	{attribute 'TcIecLibraryType'}
	{attribute 'external_name' := 'F_VN_CreateStaModel_GUID_E57A5C51_9E90_B9A1_5702_3D94CC195C09'}
	(* Create a Simplified TopoART neural network of the specified type. The initial reference count is set to one if a new model is created and kept, otherwise. Models of this type support on-line training (sample by sample), retraining, as well as scalar and vectorial predictions. It requires all input except class labels (i.e., samples and training outputs/predictions) to lie in the interval [0.0, 1.0]. The predictions of regressors need to be rescaled from the interval [0.0, 1.0] to their respective value range before usage. Depending on the parameter settings and the number of available training samples, repeated training with the same data may improve the results. Like other neural networks based on the Adaptive Resonance Theory (ART), Simplified TopoART neural networks are not prone to catastrophic inference and patricularly well-suited to incremental learning tasks. *)
	FUNCTION F_VN_CreateStaModel : HRESULT
	VAR_INPUT
		ipMlModel	:	REFERENCE TO ITcVnMlModel;	(* Returns the created model (Non-zero interface pointers are reused.) *)
		eStaType	:	ETcVnSta;	(* Simpified TopoART model type *)
		fRho	:	LREAL;	(* Vigilance parameter (controls the number of neurons that are inserted and the maximum size of the formed categories; valid range: [0.0, 1.0]; suggested range: [0.8, 1.0)) *)
		hrPrev	:	HRESULT;	(* HRESULT indicating the result of previous operations (If SUCCEEDED(hrPrev) equals false, no operation is executed.) *)
	END_VAR

END_FUNCTION

// Functions/Machine Learning/F_VN_CreateStaModelExp

	{attribute 'TcIecLibraryType'}
	{attribute 'external_name' := 'F_VN_CreateStaModelExp_GUID_8BD6F583_6D68_B761_42B8_60DD8485D486'}
	(* Create a Simplified TopoART neural network of the specified type. The initial reference count is set to one if a new model is created and kept, otherwise. Models of this type support on-line training (sample by sample), retraining, as well as scalar and vectorial predictions. It requires all input except class labels (i.e., samples and training outputs/predictions) to lie in the interval [0.0, 1.0]. The predictions of regressors need to be rescaled from the interval [0.0, 1.0] to their respective value range before usage. Depending on the parameter settings and the number of available training samples, repeated training with the same data may improve the results. Like other neural networks based on the Adaptive Resonance Theory (ART), Simplified TopoART neural networks are not prone to catastrophic inference and patricularly well-suited to incremental learning tasks. (expert function) *)
	FUNCTION F_VN_CreateStaModelExp : HRESULT
	VAR_INPUT
		ipMlModel	:	REFERENCE TO ITcVnMlModel;	(* Returns the created model (Non-zero interface pointers are reused.) *)
		eStaType	:	ETcVnSta;	(* Simpified TopoART model type *)
		fRho	:	LREAL;	(* Vigilance parameter (controls the number of neurons that are inserted and the maximum size of the formed categories; valid range: [0.0, 1.0]; suggested range: [0.8, 1.0)) *)
		nNu	:	UDINT;	(* Number of neurons used for classification and prediction (must be larger than or equal to 1; suggested range: [1, 10); default: 3) *)
		bDoublePrecision	:	BOOL;	(* If true, the model is generated with double precision (LREAL) instead of single precision (REAL). (default: FALSE) *)
		hrPrev	:	HRESULT;	(* HRESULT indicating the result of previous operations (If SUCCEEDED(hrPrev) equals false, no operation is executed.) *)
	END_VAR

END_FUNCTION

// Functions/Machine Learning/F_VN_CreateStaModelExp2

	{attribute 'TcIecLibraryType'}
	{attribute 'external_name' := 'F_VN_CreateStaModelExp2_GUID_374514C7_49DC_B14C_5A87_3ADAC4837261'}
	(* Create a Simplified TopoART neural network of the specified type. The initial reference count is set to one if a new model is created and kept, otherwise. Models of this type support on-line training (sample by sample), retraining, as well as scalar and vectorial predictions. It requires all input except class labels (i.e., samples and training outputs/predictions) to lie in the interval [0.0, 1.0]. The predictions of regressors need to be rescaled from the interval [0.0, 1.0] to their respective value range before usage. Depending on the parameter settings and the number of available training samples, repeated training with the same data may improve the results. Like other neural networks based on the Adaptive Resonance Theory (ART), Simplified TopoART neural networks are not prone to catastrophic inference and patricularly well-suited to incremental learning tasks. (additional expert function providing parameters for fine-tuning and noise reduction) *)
	FUNCTION F_VN_CreateStaModelExp2 : HRESULT
	VAR_INPUT
		ipMlModel	:	REFERENCE TO ITcVnMlModel;	(* Returns the created model (Non-zero interface pointers are reused.) *)
		eStaType	:	ETcVnSta;	(* Simpified TopoART model type *)
		fRho	:	LREAL;	(* Vigilance parameter (controls the number of neurons that are inserted and the maximum size of the formed categories; valid range: [0.0, 1.0]; suggested range: [0.8, 1.0)) *)
		nNu	:	UDINT;	(* Number of neurons used for classification and prediction (must be larger than or equal to 1; suggested range: [1, 10); default: 3) *)
		bDoublePrecision	:	BOOL;	(* If true, the model is generated with double precision (LREAL) instead of single precision (REAL). (default: FALSE) *)
		fBetaSbm	:	LREAL;	(* Learning rate of the second best-matching neuron (learning the second best-matching neuron keeps related categories closer together and might improve the results but may require a higher number of neurons and training runs; a value of 0.0 disables learning of the second best-matching neuron; valid range: [0.0, 1.0]; suggested range: [0.0, 0.5]); default: 0.0 *)
		nPhi	:	UDINT;	(* Number of samples a neuron must have learnt to become permanent (required for noise reduction; works in conjunction with nTau; must be larger than or equal to 1; higher values intensify noise reduction; a value of 1 disables removal of neuron candidates; default: 1) *)
		nTau	:	UDINT;	(* Number of learning steps after which node removal is performed (required for noise reduction; works in conjunction with nPhi; must be large enough to allow neuron candidates representing non-noise samples to become the best-matching neuron at least nPhi times before node removal; default: 100) *)
		hrPrev	:	HRESULT;	(* HRESULT indicating the result of previous operations (If SUCCEEDED(hrPrev) equals false, no operation is executed.) *)
	END_VAR

END_FUNCTION

// Functions/Machine Learning/F_VN_CreateSvmModel

	{attribute 'TcIecLibraryType'}
	{attribute 'external_name' := 'F_VN_CreateSvmModel_GUID_8D17BE1A_260C_B8D5_796F_11D521846FD9'}
	(* Create an SVM model of the specified type. The initial reference count is set to one if a new model is created and kept, otherwise. Models of this type neither support on-line training (sample by sample) nor retraining. Predictions can only be scalar. *)
	FUNCTION F_VN_CreateSvmModel : HRESULT
	VAR_INPUT
		ipMlModel	:	REFERENCE TO ITcVnMlModel;	(* Returns the created model (Non-zero interface pointers are reused.) *)
		eSvmType	:	ETcVnSvm;	(* SVM model type *)
		fC	:	LREAL;	(* Parameter C (required for TCVN_SVM_C_CLASSIFIER, TCVN_SVM_EPS_REGRESSOR, and TCVN_SVM_NU_REGRESSOR; ignored otherwise) *)
		fNu	:	LREAL;	(* Parameter nu (required for TCVN_SVM_NU_CLASSIFIER, TCVN_SVM_NOVELTY_DETECTOR, and TCVN_SVM_NU_REGRESSOR; ignored otherwise) *)
		fP	:	LREAL;	(* Parameter p (required for TCVN_SVM_EPS_REGRESSOR; ignored otherwise) *)
		eKernelType	:	ETcVnSvmKernelType;	(* Kernel type *)
		fGamma	:	LREAL;	(* Parameter gamma (used by polynomial, RBF, sigmoid, and chi-squared kernels; ignored otherwise) *)
		fCoef0	:	LREAL;	(* parameter coef0 (used by polynomial and sigmoid kernels; ignored otherwise) *)
		fDegree	:	LREAL;	(* Degree (used by polynomial kernels; ignored otherwise) *)
		hrPrev	:	HRESULT;	(* HRESULT indicating the result of previous operations (If SUCCEEDED(hrPrev) equals false, no operation is executed.) *)
	END_VAR

END_FUNCTION

// Functions/Machine Learning/F_VN_CreateSvmModelExp

	{attribute 'TcIecLibraryType'}
	{attribute 'external_name' := 'F_VN_CreateSvmModelExp_GUID_80022415_75F2_B05A_48A0_04DE64383B9C'}
	(* Create an SVM model of the specified type. The initial reference count is set to one if a new model is created and kept, otherwise. Models of this type neither support on-line training (sample by sample) nor retraining. Predictions can only be scalar. (expert function) *)
	FUNCTION F_VN_CreateSvmModelExp : HRESULT
	VAR_INPUT
		ipMlModel	:	REFERENCE TO ITcVnMlModel;	(* Returns the created model (Non-zero interface pointers are reused.) *)
		eSvmType	:	ETcVnSvm;	(* SVM model type *)
		fC	:	LREAL;	(* Parameter C (required for TCVN_SVM_C_CLASSIFIER, TCVN_SVM_EPS_REGRESSOR, and TCVN_SVM_NU_REGRESSOR; ignored otherwise) *)
		fNu	:	LREAL;	(* Parameter nu (required for TCVN_SVM_NU_CLASSIFIER, TCVN_SVM_NOVELTY_DETECTOR, and TCVN_SVM_NU_REGRESSOR; ignored otherwise) *)
		fP	:	LREAL;	(* Parameter p (required for TCVN_SVM_EPS_REGRESSOR; ignored otherwise) *)
		eKernelType	:	ETcVnSvmKernelType;	(* Kernel type *)
		fGamma	:	LREAL;	(* Parameter gamma (used by polynomial, RBF, sigmoid, and chi-squared kernels; ignored otherwise) *)
		fCoef0	:	LREAL;	(* Parameter coef0 (used by polynomial and sigmoid kernels; ignored otherwise) *)
		fDegree	:	LREAL;	(* Degree (used by polynomial kernels; ignored otherwise) *)
		nMaxIterations	:	UDINT;	(* Maximum number of iterations (disabled if it equals 0 and fEpsilon is different from 0.0; triggers the usage of the default value of 100000 if nMaxIterations and fEpsilon equal 0) *)
		fEpsilon	:	LREAL;	(* Maximum allowed difference of the error between two successive iterations (disabled if it equals 0.0 and nMaxIterations is different from 0; triggers the usage of the default value of 0.00001 if nMaxIterations and fEpsilon equal 0) *)
		hrPrev	:	HRESULT;	(* HRESULT indicating the result of previous operations (If SUCCEEDED(hrPrev) equals false, no operation is executed.) *)
	END_VAR

END_FUNCTION

// Functions/Machine Learning/F_VN_CreateSvmModelExp2

	{attribute 'TcIecLibraryType'}
	{attribute 'external_name' := 'F_VN_CreateSvmModelExp2_GUID_84CA59A5_8507_BAA1_5BD6_0739A483F2C9'}
	(* Create an SVM model of the specified type. The initial reference count is set to one if a new model is created and kept, otherwise. Models of this type neither support on-line training (sample by sample) nor retraining. Predictions can only be scalar. (additional expert function for C support vector classifiers) *)
	FUNCTION F_VN_CreateSvmModelExp2 : HRESULT
	VAR_INPUT
		ipMlModel	:	REFERENCE TO ITcVnMlModel;	(* Returns the created model (Non-zero interface pointers are reused.) *)
		eSvmType	:	ETcVnSvm;	(* SVM model type *)
		fC	:	LREAL;	(* Parameter C (required for TCVN_SVM_C_CLASSIFIER, TCVN_SVM_EPS_REGRESSOR, and TCVN_SVM_NU_REGRESSOR; ignored otherwise) *)
		fNu	:	LREAL;	(* Parameter nu (required for TCVN_SVM_NU_CLASSIFIER, TCVN_SVM_NOVELTY_DETECTOR, and TCVN_SVM_NU_REGRESSOR; ignored otherwise) *)
		fP	:	LREAL;	(* Parameter p (required for TCVN_SVM_EPS_REGRESSOR; ignored otherwise) *)
		eKernelType	:	ETcVnSvmKernelType;	(* Kernel type *)
		fGamma	:	LREAL;	(* Parameter gamma (used by polynomial, RBF, sigmoid, and chi-squared kernels; ignored otherwise) *)
		fCoef0	:	LREAL;	(* Parameter coef0 (used by polynomial and sigmoid kernels; ignored otherwise) *)
		fDegree	:	LREAL;	(* Degree (used by polynomial kernels; ignored otherwise) *)
		nMaxIterations	:	UDINT;	(* Maximum number of iterations (disabled if it equals 0 and fEpsilon is different from 0.0; triggers the usage of the default value of 100000 if nMaxIterations and fEpsilon equal 0) *)
		fEpsilon	:	LREAL;	(* Maximum allowed difference of the error between two successive iterations (disabled if it equals 0.0 and nMaxIterations is different from 0; triggers the usage of the default value of 0.00001 if nMaxIterations and fEpsilon equal 0) *)
		ipClassWeights	:	ITcVnContainer;	(* Class weights (ContainerType_Vector_REAL or ContainerType_Vector_LREAL; only valid if eSvmType equals TCVN_SVM_C_CLASSIFIER; optional, set to 0 if not required or not allowed; default: 0) *)
		hrPrev	:	HRESULT;	(* HRESULT indicating the result of previous operations (If SUCCEEDED(hrPrev) equals false, no operation is executed.) *)
	END_VAR

END_FUNCTION

// Functions/Machine Learning/F_VN_CreateSvmSgdClassifier

	{attribute 'TcIecLibraryType'}
	{attribute 'external_name' := 'F_VN_CreateSvmSgdClassifier_GUID_22F18F98_6803_BC91_601C_6D905DB53F12'}
	(* Create a linear SVM classifier using stochastic gradient descent for training. The initial reference count is set to one if a new model is created and kept, otherwise. This SVM classifier is only applicable to binary classification problems. It learns a separating hyperplane between a class with label -1 and a class with label 1. These class labels are predefined. For training, any positive class labels are mapped to 1 and any negative class labels are mapped to -1. Models of this type neither support on-line training (sample by sample) nor retraining. *)
	FUNCTION F_VN_CreateSvmSgdClassifier : HRESULT
	VAR_INPUT
		ipMlModel	:	REFERENCE TO ITcVnMlModel;	(* Returns the created model (Non-zero interface pointers are reused.) *)
		hrPrev	:	HRESULT;	(* HRESULT indicating the result of previous operations (If SUCCEEDED(hrPrev) equals false, no operation is executed.) *)
	END_VAR

END_FUNCTION

// Functions/Machine Learning/F_VN_CreateSvmSgdClassifierExp

	{attribute 'TcIecLibraryType'}
	{attribute 'external_name' := 'F_VN_CreateSvmSgdClassifierExp_GUID_DE6E86CE_13B3_BF4B_4F7F_D5DFEC535232'}
	(* Create a linear SVM classifier using stochastic gradient descent for training. The initial reference count is set to one if a new model is created and kept, otherwise. This SVM classifier is only applicable to binary classification problems. It learns a separating hyperplane between a class with label -1 and a class with label 1. These class labels are predefined. For training, any positive class labels are mapped to 1 and any negative class labels are mapped to -1. Models of this type neither support on-line training (sample by sample) nor retraining. (expert function) *)
	FUNCTION F_VN_CreateSvmSgdClassifierExp : HRESULT
	VAR_INPUT
		ipMlModel	:	REFERENCE TO ITcVnMlModel;	(* Returns the created model (Non-zero interface pointers are reused.) *)
		eType	:	ETcVnSvmSgdClassifierType;	(* Learning algorithm type (default: TCVN_SSCT_ASGD) *)
		eMarginType	:	ETcVnSvmSgdClassifierMarginType;	(* Margin type (default: TCVN_SSCMT_SOFT_MARGIN) *)
		fMarginRegularization	:	REAL;	(* Margin regularization parameter (default: 0.00001) *)
		fInitialStepSize	:	REAL;	(* Initial step size (default: 0.05) *)
		fStepDecreasingPower	:	REAL;	(* Power parameter (default: 0.75) *)
		nMaxIterations	:	UDINT;	(* Maximum number of iterations (disabled if it equals 0 and fEpsilon is different from 0.0; triggers the usage of the default value of 100000 if nMaxIterations and fEpsilon equal 0) *)
		fEpsilon	:	LREAL;	(* Maximum allowed difference of the error between two successive iterations (disabled if it equals 0.0 and nMaxIterations is different from 0; triggers the usage of the default value of 0.00001 if nMaxIterations and fEpsilon equal 0) *)
		hrPrev	:	HRESULT;	(* HRESULT indicating the result of previous operations (If SUCCEEDED(hrPrev) equals false, no operation is executed.) *)
	END_VAR

END_FUNCTION

// Functions/Machine Learning/F_VN_FeatureTransform

	{attribute 'TcIecLibraryType'}
	{attribute 'external_name' := 'F_VN_FeatureTransform_GUID_2D180149_1314_B2CD_6D03_B45D7BAFFB33'}
	(* Apply a feature transform to one or more sample(s). *)
	FUNCTION F_VN_FeatureTransform : HRESULT
	VAR_INPUT
		ipFeatureTransform	:	ITcVnMlModel;	(* Feature transform instance to be used *)
		ipSamples	:	ITcUnknown;	(* Container holding one or more of input sample(s) (ContainerType_Vector_REAL, ContainerType_Vector_LREAL, ContainerType_Vector_Vector_REAL, or ContainerType_Vector_Vector_LREAL) *)
		pipTransformed	:	POINTER TO ITcUnknown;	(* Returns the transformed sample(s) using the same type like ipSamples *)
		hrPrev	:	HRESULT;	(* HRESULT indicating the result of previous operations (If SUCCEEDED(hrPrev) equals false, no operation is executed.) *)
	END_VAR

END_FUNCTION

// Functions/Machine Learning/F_VN_GetBatchClusters

	{attribute 'TcIecLibraryType'}
	{attribute 'external_name' := 'F_VN_GetBatchClusters_GUID_B991822A_20BF_BAE1_5901_CECBAF3E4795'}
	(* Get the IDs of the best-matching clusters of a batch of samples. *)
	FUNCTION F_VN_GetBatchClusters : HRESULT
	VAR_INPUT
		ipClusterer	:	ITcVnMlModel;	(* Clusterer to be used *)
		ipSamples	:	ITcUnknown;	(* Container holding a batch of input samples (ContainerType_Vector_Vector_REAL or ContainerType_Vector_Vector_LREAL) *)
		ipClusters	:	REFERENCE TO ITcVnContainer;	(* Returns the cluster IDs (ContainerType_Vector_DINT) *)
		hrPrev	:	HRESULT;	(* HRESULT indicating the result of previous operations (If SUCCEEDED(hrPrev) equals false, no operation is executed.) *)
	END_VAR

END_FUNCTION

// Functions/Machine Learning/F_VN_GetBatchClustersExp

	{attribute 'TcIecLibraryType'}
	{attribute 'external_name' := 'F_VN_GetBatchClustersExp_GUID_01381543_FF2C_BDB4_623D_753D989F9781'}
	(* Get the IDs of the best-matching clusters of a batch of samples. *)
	FUNCTION F_VN_GetBatchClustersExp : HRESULT
	VAR_INPUT
		ipClusterer	:	ITcVnMlModel;	(* Clusterer to be used *)
		ipSamples	:	ITcUnknown;	(* Container holding a batch of input samples (ContainerType_Vector_Vector_REAL or ContainerType_Vector_Vector_LREAL) *)
		ipClusters	:	REFERENCE TO ITcVnContainer;	(* Returns the cluster IDs (ContainerType_Vector_DINT) *)
		ipNovelties	:	REFERENCE TO ITcVnContainer;	(* Returns the degree of novelty (0.0 if a sample is completely known; > 0.0 otherwise) of each sample (ContainerType_Vector_REAL; optional, set to 0 if not required) *)
		hrPrev	:	HRESULT;	(* HRESULT indicating the result of previous operations (If SUCCEEDED(hrPrev) equals false, no operation is executed.) *)
	END_VAR

END_FUNCTION

// Functions/Machine Learning/F_VN_GetBatchNovelties

	{attribute 'TcIecLibraryType'}
	{attribute 'external_name' := 'F_VN_GetBatchNovelties_GUID_97240524_1B64_B7E2_556C_1ACF30F41F39'}
	(* Get the degree of novelty of multiple samples. *)
	FUNCTION F_VN_GetBatchNovelties : HRESULT
	VAR_INPUT
		ipNoveltyDetector	:	ITcVnMlModel;	(* Novelty detector to be used *)
		ipSamples	:	ITcUnknown;	(* Container holding a batch of input samples (ContainerType_Vector_Vector_REAL or ContainerType_Vector_Vector_LREAL) *)
		ipNovelties	:	REFERENCE TO ITcVnContainer;	(* Returns the degree of novelty (0.0 if a sample is completely known; > 0.0 otherwise) of each sample (ContainerType_Vector_REAL) *)
		hrPrev	:	HRESULT;	(* HRESULT indicating the result of previous operations (If SUCCEEDED(hrPrev) equals false, no operation is executed.) *)
	END_VAR

END_FUNCTION

// Functions/Machine Learning/F_VN_GetClusterCenter

	{attribute 'TcIecLibraryType'}
	{attribute 'external_name' := 'F_VN_GetClusterCenter_GUID_E4931504_8DC6_B6D3_5D5D_2EFA9234F477'}
	(* Get the center of a cluster. *)
	FUNCTION F_VN_GetClusterCenter : HRESULT
	VAR_INPUT
		ipClusterer	:	ITcVnMlModel;	(* Clusterer to be used *)
		nCluster	:	DINT;	(* Cluster ID of the cluster the center of which is requested *)
		ipCenter	:	REFERENCE TO ITcVnContainer;	(* Returns the cluster center (ContainerType_Vector_REAL or ContainerType_Vector_LREAL depending on the floating point type internally used by the clusterer) *)
		hrPrev	:	HRESULT;	(* HRESULT indicating the result of previous operations (If SUCCEEDED(hrPrev) equals false, no operation is executed.) *)
	END_VAR

END_FUNCTION

// Functions/Machine Learning/F_VN_GetClusterNum

	{attribute 'TcIecLibraryType'}
	{attribute 'external_name' := 'F_VN_GetClusterNum_GUID_BF90D70E_F34B_BD2C_7F4D_80A10CF6A5F4'}
	(* Get the number of clusters used by this clusterer. *)
	FUNCTION F_VN_GetClusterNum : HRESULT
	VAR_INPUT
		ipClusterer	:	ITcVnMlModel;	(* Clusterer to be used *)
	END_VAR
	VAR_IN_OUT
		nClusterNum	:	ULINT;	(* Returns the number of clusters *)
	END_VAR
	VAR_INPUT
		hrPrev	:	HRESULT;	(* HRESULT indicating the result of previous operations (If SUCCEEDED(hrPrev) equals false, no operation is executed.) *)
	END_VAR

END_FUNCTION

// Functions/Machine Learning/F_VN_GetFeatureScales

	{attribute 'TcIecLibraryType'}
	{attribute 'external_name' := 'F_VN_GetFeatureScales_GUID_152933F4_9817_B6E4_5FDD_5FA5A50599FB'}
	(* Calculate the scaling parameters for each feature in the input samples based on the scaling type. *)
	FUNCTION F_VN_GetFeatureScales : HRESULT
	VAR_INPUT
		ipSamples	:	ITcVnContainer;	(* Container holding input sample(s) (ContainerType_Vector_REAL, ContainerType_Vector_LREAL, ContainerType_Vector_Vector_REAL or ContainerType_Vector_Vector_LREAL) *)
		ipScales	:	REFERENCE TO ITcVnContainer;	(* Returns a container with the scaling parameters for each feature (Vector_REAL or Vector_LREAL depending on the type of ipSamples). *)
		eFeatureScalingType	:	ETcVnFeatureScalingType;	(* Feature scaling type *)
		hrPrev	:	HRESULT;	(* HRESULT indicating the result of previous operations (If SUCCEEDED(hrPrev) equals false, no operation is executed.) *)
	END_VAR

END_FUNCTION

// Functions/Machine Learning/F_VN_GetSampleCluster

	{attribute 'TcIecLibraryType'}
	{attribute 'external_name' := 'F_VN_GetSampleCluster_GUID_D9EDADE6_09DF_BF79_401D_9EFAF11AC262'}
	(* Get the ID of the best-matching cluster of a single sample. *)
	FUNCTION F_VN_GetSampleCluster : HRESULT
	VAR_INPUT
		ipClusterer	:	ITcVnMlModel;	(* Clusterer to be used *)
		ipSample	:	ITcUnknown;	(* Container holding a single input sample (ContainerType_Vector_REAL or ContainerType_Vector_LREAL) *)
	END_VAR
	VAR_IN_OUT
		nCluster	:	DINT;	(* Returns the ID of the cluster the sample has been assigned to *)
	END_VAR
	VAR_INPUT
		hrPrev	:	HRESULT;	(* HRESULT indicating the result of previous operations (If SUCCEEDED(hrPrev) equals false, no operation is executed.) *)
	END_VAR

END_FUNCTION

// Functions/Machine Learning/F_VN_GetSampleClusterExp

	{attribute 'TcIecLibraryType'}
	{attribute 'external_name' := 'F_VN_GetSampleClusterExp_GUID_DF68DB58_441A_B462_5F9C_8B8B5A8B453F'}
	(* Get the ID of the best-matching cluster of a single sample. (expert function) *)
	FUNCTION F_VN_GetSampleClusterExp : HRESULT
	VAR_INPUT
		ipClusterer	:	ITcVnMlModel;	(* Clusterer to be used *)
		ipSample	:	ITcUnknown;	(* Container holding a single input sample (ContainerType_Vector_REAL or ContainerType_Vector_LREAL) *)
	END_VAR
	VAR_IN_OUT
		nCluster	:	DINT;	(* Returns the ID of the cluster the sample has been assigned to *)
	END_VAR
	VAR_INPUT
		fNovelty	:	REFERENCE TO REAL;	(* Returns the degree of novelty (0.0 if a sample is completely known; > 0.0 otherwise) of the presented sample (optional, set to 0 if not required) *)
		hrPrev	:	HRESULT;	(* HRESULT indicating the result of previous operations (If SUCCEEDED(hrPrev) equals false, no operation is executed.) *)
	END_VAR

END_FUNCTION

// Functions/Machine Learning/F_VN_GetSampleNovelty

	{attribute 'TcIecLibraryType'}
	{attribute 'external_name' := 'F_VN_GetSampleNovelty_GUID_39A873D6_D903_BC16_5D0D_1737EA55271D'}
	(* Get the degree of novelty of a single sample. *)
	FUNCTION F_VN_GetSampleNovelty : HRESULT
	VAR_INPUT
		ipNoveltyDetector	:	ITcVnMlModel;	(* Novelty detector to be used *)
		ipSample	:	ITcUnknown;	(* Container holding a single input sample (ContainerType_Vector_REAL or ContainerType_Vector_LREAL) *)
	END_VAR
	VAR_IN_OUT
		fNovelty	:	REAL;	(* Returns the degree of novelty (0.0 if a sample is completely known; > 0.0 otherwise) of the presented sample *)
	END_VAR
	VAR_INPUT
		hrPrev	:	HRESULT;	(* HRESULT indicating the result of previous operations (If SUCCEEDED(hrPrev) equals false, no operation is executed.) *)
	END_VAR

END_FUNCTION

// Functions/Machine Learning/F_VN_InverseFeatureScaling

	{attribute 'TcIecLibraryType'}
	{attribute 'external_name' := 'F_VN_InverseFeatureScaling_GUID_FE8FDE22_64A6_B82E_5950_09F49A4CC796'}
	(* Apply the inverse of feature scaling to one or more sample(s). *)
	FUNCTION F_VN_InverseFeatureScaling : HRESULT
	VAR_INPUT
		ipSamples	:	ITcVnContainer;	(* Container holding one or more input sample(s) (ContainerType_Vector_REAL, ContainerType_Vector_LREAL, ContainerType_Vector_Vector_REAL, or ContainerType_Vector_Vector_LREAL) *)
		ipScales	:	ITcVnContainer;	(* Container with the scaling parameters of each feature (type ContainerType_Vector_REAL or ContainerType_Vector_LREAL). *)
		ipInverseSamples	:	REFERENCE TO ITcVnContainer;	(* Returns the inversed sample(s) using the scaling type and parameters of ipScales. It has the same type of ipSamples. If the same container ipSamples is used, the source data will be replaced. *)
		hrPrev	:	HRESULT;	(* HRESULT indicating the result of previous operations (If SUCCEEDED(hrPrev) equals false, no operation is executed.) *)
	END_VAR

END_FUNCTION

// Functions/Machine Learning/F_VN_InverseFeatureScaling_REAL

	{attribute 'TcIecLibraryType'}
	{attribute 'external_name' := 'F_VN_InverseFeatureScaling_REAL_GUID_1201C1F8_7D25_B625_41FC_0E90A3247281'}
	(* Apply the inverse of feature scaling to a single value. *)
	FUNCTION F_VN_InverseFeatureScaling_REAL : HRESULT
	VAR_INPUT
		fSample	:	REAL;	(* Sample value *)
		ipScales	:	ITcVnContainer;	(* Container with the scaling parameters of each feature (type ContainerType_Vector_REAL or ContainerType_Vector_LREAL). *)
	END_VAR
	VAR_IN_OUT
		fInverseSample	:	REAL;	(* Returns the inversed sample. *)
	END_VAR
	VAR_INPUT
		hrPrev	:	HRESULT;	(* HRESULT indicating the result of previous operations (If SUCCEEDED(hrPrev) equals false, no operation is executed.) *)
	END_VAR

END_FUNCTION

// Functions/Machine Learning/F_VN_InverseFeatureScalingExp

	{attribute 'TcIecLibraryType'}
	{attribute 'external_name' := 'F_VN_InverseFeatureScalingExp_GUID_6011A69B_BC3C_B4AD_6BA0_0FF48B427FDA'}
	(* Apply the inverse of feature scaling to one or more sample(s). [fA, fB] should be used if the scaling has been performed using TCVN_FST1_MINMAX with a predetermined output range.. (expert function) *)
	FUNCTION F_VN_InverseFeatureScalingExp : HRESULT
	VAR_INPUT
		ipSamples	:	ITcVnContainer;	(* Container holding one or more input sample(s) (ContainerType_Vector_REAL, ContainerType_Vector_LREAL, ContainerType_Vector_Vector_REAL, or ContainerType_Vector_Vector_LREAL) *)
		ipScales	:	ITcVnContainer;	(* Container with the scaling parameters of each feature (type ContainerType_Vector_REAL or ContainerType_Vector_LREAL). *)
		ipInverseSamples	:	REFERENCE TO ITcVnContainer;	(* Returns the inversed sample(s) using the scaling type and parameters of ipScales. It has the same type of ipSamples. If the same container ipSamples is used, the source data will be replaced. *)
		fA	:	LREAL;	(* represents the lower bound of the range for TCVN_FST1_MINMAX *)
		fB	:	LREAL;	(* represents the upper bound of the range for TCVN_FST1_MINMAX *)
		hrPrev	:	HRESULT;	(* HRESULT indicating the result of previous operations (If SUCCEEDED(hrPrev) equals false, no operation is executed.) *)
	END_VAR

END_FUNCTION

// Functions/Machine Learning/F_VN_InverseFeatureScalingExp_REAL

	{attribute 'TcIecLibraryType'}
	{attribute 'external_name' := 'F_VN_InverseFeatureScalingExp_REAL_GUID_C9B73D36_4564_B6F0_65B6_270F53192161'}
	(* Apply the inverse of feature scaling to a single value. [fA, fB] should be used if the scaling has been performed using TCVN_FST1_MINMAX with a predetermined output range. *)
	FUNCTION F_VN_InverseFeatureScalingExp_REAL : HRESULT
	VAR_INPUT
		fSample	:	REAL;	(* Sample value *)
		ipScales	:	ITcVnContainer;	(* Container with the scaling parameters of each feature (type ContainerType_Vector_REAL or ContainerType_Vector_LREAL). *)
	END_VAR
	VAR_IN_OUT
		fInverseSample	:	REAL;	(* Returns the inversed sample. *)
	END_VAR
	VAR_INPUT
		fA	:	LREAL;	(* represents the lower bound of the range for TCVN_FST1_MINMAX *)
		fB	:	LREAL;	(* represents the upper bound of the range for TCVN_FST1_MINMAX *)
		hrPrev	:	HRESULT;	(* HRESULT indicating the result of previous operations (If SUCCEEDED(hrPrev) equals false, no operation is executed.) *)
	END_VAR

END_FUNCTION

// Functions/Machine Learning/F_VN_InverseFeatureTransform

	{attribute 'TcIecLibraryType'}
	{attribute 'external_name' := 'F_VN_InverseFeatureTransform_GUID_36FA6EBF_2E20_B057_4C4D_1F432CD52CC5'}
	(* Apply an inverse feature transform to one or more sample(s). *)
	FUNCTION F_VN_InverseFeatureTransform : HRESULT
	VAR_INPUT
		ipFeatureTransform	:	ITcVnMlModel;	(* Feature transform instance to be used *)
		ipSamples	:	ITcUnknown;	(* Container holding one or more of input sample(s) (ContainerType_Vector_REAL, ContainerType_Vector_LREAL, ContainerType_Vector_Vector_REAL, or ContainerType_Vector_Vector_LREAL) *)
		pipTransformed	:	POINTER TO ITcUnknown;	(* Returns the transformed sample(s) using the same type like ipSamples *)
		hrPrev	:	HRESULT;	(* HRESULT indicating the result of previous operations (If SUCCEEDED(hrPrev) equals false, no operation is executed.) *)
	END_VAR

END_FUNCTION

// Functions/Machine Learning/F_VN_PredictBatch

	{attribute 'TcIecLibraryType'}
	{attribute 'external_name' := 'F_VN_PredictBatch_GUID_7D6AF5D3_F545_BA81_6792_DBF8D05FF13D'}
	(* Compute predictions for a batch of samples. *)
	FUNCTION F_VN_PredictBatch : HRESULT
	VAR_INPUT
		ipMlModel	:	ITcVnMlModel;	(* Classifier or regressor to be used *)
		ipSamples	:	ITcUnknown;	(* Container holding a batch of input samples (ContainerType_Vector_Vector_REAL or ContainerType_Vector_Vector_LREAL) *)
		ipPredictions	:	REFERENCE TO ITcVnContainer;	(* Returns the predicted outputs (depending on ipSamples; class labels (for classification, ContainerType_Vector_DINT) or real-valued predictions (for regression with scalar output, ContainerType_Vector_REAL or ContainerType_Vector_LREAL; for regression with vectorial output, ContainerType_Vector_Vector_REAL or ContainerType_Vector_Vector_LREAL)) *)
		hrPrev	:	HRESULT;	(* HRESULT indicating the result of previous operations (If SUCCEEDED(hrPrev) equals false, no operation is executed.) *)
	END_VAR

END_FUNCTION

// Functions/Machine Learning/F_VN_PredictBatchExp

	{attribute 'TcIecLibraryType'}
	{attribute 'external_name' := 'F_VN_PredictBatchExp_GUID_C38FEE18_09F7_BE98_52DE_06033125E4BC'}
	(* Compute predictions for a batch of samples. (expert function) *)
	FUNCTION F_VN_PredictBatchExp : HRESULT
	VAR_INPUT
		ipMlModel	:	ITcVnMlModel;	(* Classifier or regressor to be used *)
		ipSamples	:	ITcUnknown;	(* Container holding a batch of input samples (ContainerType_Vector_Vector_REAL or ContainerType_Vector_Vector_LREAL) *)
		ipPredictions	:	REFERENCE TO ITcVnContainer;	(* Returns the predicted outputs (depending on ipSamples; class labels (for classification, ContainerType_Vector_DINT) or real-valued predictions (for regression with scalar output, ContainerType_Vector_REAL or ContainerType_Vector_LREAL; for regression with vectorial output, ContainerType_Vector_Vector_REAL or ContainerType_Vector_Vector_LREAL)) *)
		ipNovelties	:	REFERENCE TO ITcVnContainer;	(* Returns the degree of novelty (0.0 if a sample is completely known; > 0.0 otherwise) of each sample (ContainerType_Vector_REAL; optional, set to 0 if not required) *)
		hrPrev	:	HRESULT;	(* HRESULT indicating the result of previous operations (If SUCCEEDED(hrPrev) equals false, no operation is executed.) *)
	END_VAR

END_FUNCTION

// Functions/Machine Learning/F_VN_PredictSampleClass

	{attribute 'TcIecLibraryType'}
	{attribute 'external_name' := 'F_VN_PredictSampleClass_GUID_4E1D7695_AD53_B95E_78AD_1EE49BFC5C71'}
	(* Classify a single sample. *)
	FUNCTION F_VN_PredictSampleClass : HRESULT
	VAR_INPUT
		ipClassifier	:	ITcVnMlModel;	(* Classifier to be used *)
		ipSample	:	ITcUnknown;	(* Container holding a single input sample (ContainerType_Vector_REAL or ContainerType_Vector_LREAL) *)
	END_VAR
	VAR_IN_OUT
		nClass	:	DINT;	(* Returns the classification result *)
	END_VAR
	VAR_INPUT
		hrPrev	:	HRESULT;	(* HRESULT indicating the result of previous operations (If SUCCEEDED(hrPrev) equals false, no operation is executed.) *)
	END_VAR

END_FUNCTION

// Functions/Machine Learning/F_VN_PredictSampleClassExp

	{attribute 'TcIecLibraryType'}
	{attribute 'external_name' := 'F_VN_PredictSampleClassExp_GUID_7AF8CE47_2D0D_B2AE_4405_566F1365D87E'}
	(* Classify a single sample. (expert function) *)
	FUNCTION F_VN_PredictSampleClassExp : HRESULT
	VAR_INPUT
		ipClassifier	:	ITcVnMlModel;	(* Classifier to be used *)
		ipSample	:	ITcUnknown;	(* Container holding a single input sample (ContainerType_Vector_REAL or ContainerType_Vector_LREAL) *)
	END_VAR
	VAR_IN_OUT
		nClass	:	DINT;	(* Returns the classification result *)
	END_VAR
	VAR_INPUT
		fNovelty	:	REFERENCE TO REAL;	(* Returns the degree of novelty (0.0 if a sample is completely known; > 0.0 otherwise) of the presented sample (optional, set to 0 if not required) *)
		hrPrev	:	HRESULT;	(* HRESULT indicating the result of previous operations (If SUCCEEDED(hrPrev) equals false, no operation is executed.) *)
	END_VAR

END_FUNCTION

// Functions/Machine Learning/F_VN_PredictSampleScalar

	{attribute 'TcIecLibraryType'}
	{attribute 'external_name' := 'F_VN_PredictSampleScalar_GUID_A0660891_3ED0_BD79_45C7_B847E30A9869'}
	(* Compute a scalar prediction for a single sample. *)
	FUNCTION F_VN_PredictSampleScalar : HRESULT
	VAR_INPUT
		ipRegressor	:	ITcVnMlModel;	(* Regressor to be used *)
		ipSample	:	ITcUnknown;	(* Container holding a single input sample (ContainerType_Vector_REAL or ContainerType_Vector_LREAL) *)
	END_VAR
	VAR_IN_OUT
		fPrediction	:	REAL;	(* Returns the predicted output *)
	END_VAR
	VAR_INPUT
		hrPrev	:	HRESULT;	(* HRESULT indicating the result of previous operations (If SUCCEEDED(hrPrev) equals false, no operation is executed.) *)
	END_VAR

END_FUNCTION

// Functions/Machine Learning/F_VN_PredictSampleScalarExp

	{attribute 'TcIecLibraryType'}
	{attribute 'external_name' := 'F_VN_PredictSampleScalarExp_GUID_32126386_2E2D_B430_66C6_B8A4437C5BD6'}
	(* Compute a scalar prediction for a single sample. (expert function) *)
	FUNCTION F_VN_PredictSampleScalarExp : HRESULT
	VAR_INPUT
		ipRegressor	:	ITcVnMlModel;	(* Regressor to be used *)
		ipSample	:	ITcUnknown;	(* Container holding a single input sample (ContainerType_Vector_REAL or ContainerType_Vector_LREAL) *)
	END_VAR
	VAR_IN_OUT
		fPrediction	:	REAL;	(* Returns the predicted output *)
	END_VAR
	VAR_INPUT
		fNovelty	:	REFERENCE TO REAL;	(* Returns the degree of novelty (0.0 if a sample is completely known; > 0.0 otherwise) of the presented sample (optional, set to 0 if not required) *)
		hrPrev	:	HRESULT;	(* HRESULT indicating the result of previous operations (If SUCCEEDED(hrPrev) equals false, no operation is executed.) *)
	END_VAR

END_FUNCTION

// Functions/Machine Learning/F_VN_PredictSampleVector

	{attribute 'TcIecLibraryType'}
	{attribute 'external_name' := 'F_VN_PredictSampleVector_GUID_1341F380_9576_B968_589D_54E9FDC95A1C'}
	(* Compute a vectorial prediction for a single sample. *)
	FUNCTION F_VN_PredictSampleVector : HRESULT
	VAR_INPUT
		ipRegressor	:	ITcVnMlModel;	(* Regressor to be used *)
		ipSample	:	ITcUnknown;	(* Container holding a single input sample (ContainerType_Vector_REAL or ContainerType_Vector_LREAL) *)
		ipPrediction	:	REFERENCE TO ITcVnContainer;	(* Returns the predicted output (ContainerType_Vector_REAL or ContainerType_Vector_LREAL, depending on ipSample) *)
		hrPrev	:	HRESULT;	(* HRESULT indicating the result of previous operations (If SUCCEEDED(hrPrev) equals false, no operation is executed.) *)
	END_VAR

END_FUNCTION

// Functions/Machine Learning/F_VN_PredictSampleVectorExp

	{attribute 'TcIecLibraryType'}
	{attribute 'external_name' := 'F_VN_PredictSampleVectorExp_GUID_031F0675_23FD_B293_640F_296778A8E4F6'}
	(* Compute a vectorial prediction for a single sample. (expert function) *)
	FUNCTION F_VN_PredictSampleVectorExp : HRESULT
	VAR_INPUT
		ipRegressor	:	ITcVnMlModel;	(* Regressor to be used *)
		ipSample	:	ITcUnknown;	(* Container holding a single input sample (ContainerType_Vector_REAL or ContainerType_Vector_LREAL) *)
		ipPrediction	:	REFERENCE TO ITcVnContainer;	(* Returns the predicted output (ContainerType_Vector_REAL or ContainerType_Vector_LREAL, depending on ipSample) *)
		fNovelty	:	REFERENCE TO REAL;	(* Returns the degree of novelty (0.0 if a sample is completely known; > 0.0 otherwise) of the presented sample (optional, set to 0 if not required) *)
		hrPrev	:	HRESULT;	(* HRESULT indicating the result of previous operations (If SUCCEEDED(hrPrev) equals false, no operation is executed.) *)
	END_VAR

END_FUNCTION

// Functions/Machine Learning/F_VN_FeatureScaling

	{attribute 'TcIecLibraryType'}
	{attribute 'external_name' := 'F_VN_FeatureScaling_GUID_9BD98239_4277_BFE9_7F08_2E1B5FF5F5E8'}
	(* Apply a feature scaling to one or more sample(s). *)
	FUNCTION F_VN_FeatureScaling : HRESULT
	VAR_INPUT
		ipSamples	:	ITcVnContainer;	(* Container holding one or more input sample(s) (ContainerType_Vector_REAL, ContainerType_Vector_LREAL, ContainerType_Vector_Vector_REAL, or ContainerType_Vector_Vector_LREAL) *)
		ipScales	:	ITcVnContainer;	(* Container with the scaling parameters of each feature (type ContainerType_Vector_REAL or ContainerType_Vector_LREAL). *)
		ipScaledSamples	:	REFERENCE TO ITcVnContainer;	(* Returns the scaled sample(s) using the same type like ipSamples. If the same container ipSamples is uesd, the source data will be replaced. *)
		hrPrev	:	HRESULT;	(* HRESULT indicating the result of previous operations (If SUCCEEDED(hrPrev) equals false, no operation is executed.) *)
	END_VAR

END_FUNCTION

// Functions/Machine Learning/F_VN_FeatureScalingExp

	{attribute 'TcIecLibraryType'}
	{attribute 'external_name' := 'F_VN_FeatureScalingExp_GUID_62DE1C89_F96E_B166_52C9_6230A4FA8FF4'}
	(* Apply a feature scaling to one or more sample(s) and get output range between [fA, fB] in the case of TCVN_FST1_MINMAX.  (expert function) *)
	FUNCTION F_VN_FeatureScalingExp : HRESULT
	VAR_INPUT
		ipSamples	:	ITcVnContainer;	(* Container holding one or more input sample(s) (ContainerType_Vector_REAL, ContainerType_Vector_LREAL, ContainerType_Vector_Vector_REAL, or ContainerType_Vector_Vector_LREAL) *)
		ipScales	:	ITcVnContainer;	(* Container with the scaling parameters of each feature (type ContainerType_Vector_REAL or ContainerType_Vector_LREAL). *)
		ipScaledSamples	:	REFERENCE TO ITcVnContainer;	(* Returns the scaled sample(s) using the same type like ipSamples. If the same container ipSamples is uesd, the source data will be replaced. *)
		fA	:	LREAL;	(* represents the lower bound of the range for TCVN_FST1_MINMAX *)
		fB	:	LREAL;	(* represents the upper bound of the range for TCVN_FST1_MINMAX *)
		hrPrev	:	HRESULT;	(* HRESULT indicating the result of previous operations (If SUCCEEDED(hrPrev) equals false, no operation is executed.) *)
	END_VAR

END_FUNCTION

// Functions/Machine Learning/F_VN_TrainBatch

	{attribute 'TcIecLibraryType'}
	{attribute 'external_name' := 'F_VN_TrainBatch_GUID_77947D56_1092_B041_6AD6_45459A0EDE0C'}
	(* Train a classifier, a clusterer, a novelty detector, or a regressor with a batch of samples. On-line trainable models are trained once with each sample. Depending on the application and the number of available training samples, repeated training of such models with the same data may improve the results. *)
	FUNCTION F_VN_TrainBatch : HRESULT
	VAR_INPUT
		ipMlModel	:	ITcVnMlModel;	(* Classifier, clusterer, novelty detector, or regressor to be used *)
		ipSamples	:	ITcUnknown;	(* Container holding a batch of input samples (ContainerType_Vector_Vector_REAL or ContainerType_Vector_Vector_LREAL) *)
		ipOutputs	:	ITcVnContainer;	(* Class labels (for classification, ContainerType_Vector_DINT) or target outputs (for regression with scalar output, ContainerType_Vector_REAL or ContainerType_Vector_LREAL; for regression with vectorial output, ContainerType_Vector_Vector_REAL or ContainerType_Vector_Vector_LREAL) to be learnt (must be 0 for clusterers and for novelty detectors) *)
		hrPrev	:	HRESULT;	(* HRESULT indicating the result of previous operations (If SUCCEEDED(hrPrev) equals false, no operation is executed.) *)
	END_VAR

END_FUNCTION

// Functions/Machine Learning/F_VN_TrainBatchClusters

	{attribute 'TcIecLibraryType'}
	{attribute 'external_name' := 'F_VN_TrainBatchClusters_GUID_23468B3D_3C92_B481_59BE_FD8A5A9CA9B1'}
	(* Train a clusterer with a batch of samples and return the IDs of the clusters the samples have been assigned to, if requested. On-line trainable clusterers are trained once with each sample. Depending on the application and the number of available training samples, repeated training of such models with the same data may improve the results. *)
	FUNCTION F_VN_TrainBatchClusters : HRESULT
	VAR_INPUT
		ipClusterer	:	ITcVnMlModel;	(* Clusterer to be used *)
		ipSamples	:	ITcUnknown;	(* Container holding a batch of input samples (ContainerType_Vector_Vector_REAL or ContainerType_Vector_Vector_LREAL) *)
		ipClusters	:	REFERENCE TO ITcVnContainer;	(* Returns the IDs of the clusters the samples have been assigned to (ContainerType_Vector_DINT; optional, set to 0 if not required) *)
		hrPrev	:	HRESULT;	(* HRESULT indicating the result of previous operations (If SUCCEEDED(hrPrev) equals false, no operation is executed.) *)
	END_VAR

END_FUNCTION

// Functions/Machine Learning/F_VN_TrainSample

	{attribute 'TcIecLibraryType'}
	{attribute 'external_name' := 'F_VN_TrainSample_GUID_6B0A2796_5FCD_B08B_5BD0_FF7775FE4207'}
	(* Train a clusterer or a novelty detector with a single sample. *)
	FUNCTION F_VN_TrainSample : HRESULT
	VAR_INPUT
		ipMlModel	:	ITcVnMlModel;	(* Clusterer or novelty detector to be used *)
		ipSample	:	ITcUnknown;	(* Container holding a single input sample (ContainerType_Vector_REAL or ContainerType_Vector_LREAL) *)
		hrPrev	:	HRESULT;	(* HRESULT indicating the result of previous operations (If SUCCEEDED(hrPrev) equals false, no operation is executed.) *)
	END_VAR

END_FUNCTION

// Functions/Machine Learning/F_VN_TrainSampleClass

	{attribute 'TcIecLibraryType'}
	{attribute 'external_name' := 'F_VN_TrainSampleClass_GUID_01CA19E7_3CA5_B1FA_5D6E_B93EEC8BFC95'}
	(* Train a classifier with a single sample. *)
	FUNCTION F_VN_TrainSampleClass : HRESULT
	VAR_INPUT
		ipClassifier	:	ITcVnMlModel;	(* Classifier to be used *)
		ipSample	:	ITcUnknown;	(* Container holding a single input sample (ContainerType_Vector_REAL or ContainerType_Vector_LREAL) *)
		nClass	:	DINT;	(* Class label to be learnt *)
		hrPrev	:	HRESULT;	(* HRESULT indicating the result of previous operations (If SUCCEEDED(hrPrev) equals false, no operation is executed.) *)
	END_VAR

END_FUNCTION

// Functions/Machine Learning/F_VN_TrainSampleCluster

	{attribute 'TcIecLibraryType'}
	{attribute 'external_name' := 'F_VN_TrainSampleCluster_GUID_305233B5_B709_B570_55D4_6B695278CCCF'}
	(* Train a clusterer with a single sample and return the ID of the cluster the sample has been assigned to, if requested. The clusterer must be online trainable. *)
	FUNCTION F_VN_TrainSampleCluster : HRESULT
	VAR_INPUT
		ipClusterer	:	ITcVnMlModel;	(* Clusterer to be used *)
		ipSample	:	ITcUnknown;	(* Container holding a single input sample (ContainerType_Vector_REAL or ContainerType_Vector_LREAL) *)
		nCluster	:	REFERENCE TO DINT;	(* Returns the ID of the cluster the sample has been assigned to (If the pointer is 0, no cluster ID is requested.) *)
		hrPrev	:	HRESULT;	(* HRESULT indicating the result of previous operations (If SUCCEEDED(hrPrev) equals false, no operation is executed.) *)
	END_VAR

END_FUNCTION

// Functions/Machine Learning/F_VN_TrainSampleScalar

	{attribute 'TcIecLibraryType'}
	{attribute 'external_name' := 'F_VN_TrainSampleScalar_GUID_58D155F2_E9EF_BEA3_57F6_8E172A1962B7'}
	(* Train a regressor with a single sample and scalar output. *)
	FUNCTION F_VN_TrainSampleScalar : HRESULT
	VAR_INPUT
		ipRegressor	:	ITcVnMlModel;	(* Regressor to be used *)
		ipSample	:	ITcUnknown;	(* Container holding a single input sample (ContainerType_Vector_REAL or ContainerType_Vector_LREAL) *)
		fOutput	:	REAL;	(* Scalar output to be learnt *)
		hrPrev	:	HRESULT;	(* HRESULT indicating the result of previous operations (If SUCCEEDED(hrPrev) equals false, no operation is executed.) *)
	END_VAR

END_FUNCTION

// Functions/Machine Learning/F_VN_TrainSampleVector

	{attribute 'TcIecLibraryType'}
	{attribute 'external_name' := 'F_VN_TrainSampleVector_GUID_A18A19AB_C46B_B59A_5A60_81FD02D259FC'}
	(* Train a regressor with a single sample and vectorial output. *)
	FUNCTION F_VN_TrainSampleVector : HRESULT
	VAR_INPUT
		ipRegressor	:	ITcVnMlModel;	(* Regressor to be used *)
		ipSample	:	ITcUnknown;	(* Container holding a single input sample (ContainerType_Vector_REAL or ContainerType_Vector_LREAL) *)
		ipOutput	:	ITcVnContainer;	(* Vectorial output to be learnt (ContainerType_Vector_REAL or ContainerType_Vector_LREAL) *)
		hrPrev	:	HRESULT;	(* HRESULT indicating the result of previous operations (If SUCCEEDED(hrPrev) equals false, no operation is executed.) *)
	END_VAR

END_FUNCTION

// Functions/Drawing/F_VN_DrawArrow

	{attribute 'TcIecLibraryType'}
	{attribute 'external_name' := 'F_VN_DrawArrow_GUID_25F3FD2E_299D_B451_64DE_CE60C6F92FCB'}
	(* Draw an arrowed line. *)
	FUNCTION F_VN_DrawArrow : HRESULT
	VAR_INPUT
		nX1	:	UDINT;	(* x coordinate of the start point *)
		nY1	:	UDINT;	(* y coordinate of the start point *)
		nX2	:	UDINT;	(* x coordinate of the end point *)
		nY2	:	UDINT;	(* y coordinate of the end point *)
		ipDestImage	:	ITcVnImage;	(* Destination image *)
	END_VAR
	VAR_IN_OUT
		aColor	:	TcVnVector4_LREAL;	(* Color *)
	END_VAR
	VAR_INPUT
		nThickness	:	DINT;	(* Line thickness *)
		bDoubleHead	:	BOOL;	(* To draw an arrow on each side of the line. *)
		hrPrev	:	HRESULT;	(* HRESULT indicating the result of previous operations (If SUCCEEDED(hrPrev) equals false, no operation is executed.) *)
	END_VAR

END_FUNCTION

// Functions/Drawing/F_VN_DrawArrow_TcVnVector4_DINT

	{attribute 'TcIecLibraryType'}
	{attribute 'external_name' := 'F_VN_DrawArrow_TcVnVector4_DINT_GUID_C9FB1724_53DB_BE4D_5F84_0D1E2B7168A9'}
	(* Draw an arrowed line. *)
	FUNCTION F_VN_DrawArrow_TcVnVector4_DINT : HRESULT
	VAR_IN_OUT
		aLine	:	TcVnVector4_DINT;	(* The start and end point of a line segment [x1, y1, x2, y2] *)
	END_VAR
	VAR_INPUT
		ipDestImage	:	ITcVnImage;	(* Destination image *)
	END_VAR
	VAR_IN_OUT
		aColor	:	TcVnVector4_LREAL;	(* Color *)
	END_VAR
	VAR_INPUT
		nThickness	:	DINT;	(* Line thickness *)
		bDoubleHead	:	BOOL;	(* To draw an arrow on each side of the line. *)
		hrPrev	:	HRESULT;	(* HRESULT indicating the result of previous operations (If SUCCEEDED(hrPrev) equals false, no operation is executed.) *)
	END_VAR

END_FUNCTION

// Functions/Drawing/F_VN_DrawArrowExp

	{attribute 'TcIecLibraryType'}
	{attribute 'external_name' := 'F_VN_DrawArrowExp_GUID_9C18B8A0_F473_BE5B_424A_0246D0DE2706'}
	(* Draws an arrowed line. (expert function) *)
	FUNCTION F_VN_DrawArrowExp : HRESULT
	VAR_INPUT
		nX1	:	UDINT;	(* x coordinate of the start point *)
		nY1	:	UDINT;	(* y coordinate of the start point *)
		nX2	:	UDINT;	(* x coordinate of the end point *)
		nY2	:	UDINT;	(* y coordinate of the end point *)
		ipDestImage	:	ITcVnImage;	(* Destination image *)
	END_VAR
	VAR_IN_OUT
		aColor	:	TcVnVector4_LREAL;	(* Color *)
	END_VAR
	VAR_INPUT
		nThickness	:	DINT;	(* Line thickness *)
		bDoubleHead	:	BOOL;	(* To draw an arrow on each side of the line. *)
		eLineType	:	ETcVnLineType;	(* Line type *)
		nShift	:	UDINT;	(* Fractional bits of the coordinates (bit shift) *)
		fTipLenght	:	LREAL;	(* Lenght of the arrow's tip as a fraction of the line's lenght *)
		hrPrev	:	HRESULT;	(* HRESULT indicating the result of previous operations (If SUCCEEDED(hrPrev) equals false, no operation is executed.) *)
	END_VAR

END_FUNCTION

// Functions/Drawing/F_VN_DrawArrowExp_TcVnVector4_DINT

	{attribute 'TcIecLibraryType'}
	{attribute 'external_name' := 'F_VN_DrawArrowExp_TcVnVector4_DINT_GUID_EF730414_30E1_B01F_5AE0_0D2C90429698'}
	(* Draws an arrowed line. (expert function) *)
	FUNCTION F_VN_DrawArrowExp_TcVnVector4_DINT : HRESULT
	VAR_IN_OUT
		aLine	:	TcVnVector4_DINT;	(* The start and end point of a line segment [x1, y1, x2, y2] *)
	END_VAR
	VAR_INPUT
		ipDestImage	:	ITcVnImage;	(* Destination image *)
	END_VAR
	VAR_IN_OUT
		aColor	:	TcVnVector4_LREAL;	(* Color *)
	END_VAR
	VAR_INPUT
		nThickness	:	DINT;	(* Line thickness *)
		bDoubleHead	:	BOOL;	(* To draw an arrow on each side of the line. *)
		eLineType	:	ETcVnLineType;	(* Line type *)
		nShift	:	UDINT;	(* Fractional bits of the coordinates (bit shift) *)
		fTipLenght	:	LREAL;	(* Lenght of the arrow's tip as a fraction of the line's lenght *)
		hrPrev	:	HRESULT;	(* HRESULT indicating the result of previous operations (If SUCCEEDED(hrPrev) equals false, no operation is executed.) *)
	END_VAR

END_FUNCTION

// Functions/Drawing/F_VN_DrawCircle

	{attribute 'TcIecLibraryType'}
	{attribute 'external_name' := 'F_VN_DrawCircle_GUID_E122AF07_4C05_B9A4_6C3D_88261C7D954A'}
	(* Draws a circle. *)
	FUNCTION F_VN_DrawCircle : HRESULT
	VAR_INPUT
		nCenterX	:	UDINT;	(* x coordinate of the center *)
		nCenterY	:	UDINT;	(* y coordinate of the center *)
		nRadius	:	UDINT;	(* Radius *)
		ipDestImage	:	ITcVnImage;	(* Destination image *)
	END_VAR
	VAR_IN_OUT
		aColor	:	TcVnVector4_LREAL;	(* Color *)
	END_VAR
	VAR_INPUT
		nThickness	:	DINT;	(* Line thickness (if negative, the circle is filled) *)
		hrPrev	:	HRESULT;	(* HRESULT indicating the result of previous operations (If SUCCEEDED(hrPrev) equals false, no operation is executed.) *)
	END_VAR

END_FUNCTION

// Functions/Drawing/F_VN_DrawCircleExp

	{attribute 'TcIecLibraryType'}
	{attribute 'external_name' := 'F_VN_DrawCircleExp_GUID_EF9D9484_62D8_B300_4669_483012B110FD'}
	(* Draws a circle. *)
	FUNCTION F_VN_DrawCircleExp : HRESULT
	VAR_INPUT
		nCenterX	:	UDINT;	(* x coordinate of the center *)
		nCenterY	:	UDINT;	(* y coordinate of the center *)
		nRadius	:	UDINT;	(* Radius *)
		ipDestImage	:	ITcVnImage;	(* Destination image *)
	END_VAR
	VAR_IN_OUT
		aColor	:	TcVnVector4_LREAL;	(* Color *)
	END_VAR
	VAR_INPUT
		nThickness	:	DINT;	(* Line thickness (if negative, the circle is filled) *)
		eLineType	:	ETcVnLineType;	(* Line type *)
		hrPrev	:	HRESULT;	(* HRESULT indicating the result of previous operations (If SUCCEEDED(hrPrev) equals false, no operation is executed.) *)
	END_VAR

END_FUNCTION

// Functions/Drawing/F_VN_DrawCircles

	{attribute 'TcIecLibraryType'}
	{attribute 'external_name' := 'F_VN_DrawCircles_GUID_1786A42B_D930_BC20_6852_A8E93EECF953'}
	(* Draws circles. *)
	FUNCTION F_VN_DrawCircles : HRESULT
	VAR_INPUT
		ipCircles	:	ITcVnContainer;	(* Container with circles (ContainerType_Vector_TcVnVector3_REAL; Each container element contains the x coordinate of the circle center [0], the y coordinate of the circle center [1], and the radius [2].) *)
		nCircleIndex	:	DINT;	(* Index of a specific circle to be drawn (if negative, all circles within the container are drawn) *)
		ipDestImage	:	ITcVnImage;	(* Destination image *)
	END_VAR
	VAR_IN_OUT
		aColor	:	TcVnVector4_LREAL;	(* Color *)
	END_VAR
	VAR_INPUT
		nThickness	:	DINT;	(* Line thickness (if negative, the circle is filled) *)
		hrPrev	:	HRESULT;	(* HRESULT indicating the result of previous operations (If SUCCEEDED(hrPrev) equals false, no operation is executed.) *)
	END_VAR

END_FUNCTION

// Functions/Drawing/F_VN_DrawCirclesExp

	{attribute 'TcIecLibraryType'}
	{attribute 'external_name' := 'F_VN_DrawCirclesExp_GUID_44E89322_C77B_BF23_6DF7_7C79B1EF5745'}
	(* Draws circles. (expert function) *)
	FUNCTION F_VN_DrawCirclesExp : HRESULT
	VAR_INPUT
		ipCircles	:	ITcVnContainer;	(* Container with circles (ContainerType_Vector_TcVnVector3_REAL; Each container element contains the x coordinate of the circle center [0], the y coordinate of the circle center [1], and the radius [2].) *)
		nCircleIndex	:	DINT;	(* Index of a specific circle to be drawn (if negative, all circles within the container are drawn) *)
		ipDestImage	:	ITcVnImage;	(* Destination image *)
	END_VAR
	VAR_IN_OUT
		aColor	:	TcVnVector4_LREAL;	(* Color *)
	END_VAR
	VAR_INPUT
		nThickness	:	DINT;	(* Line thickness (if negative, the circle is filled) *)
		eLineType	:	ETcVnLineType;	(* Line type *)
		hrPrev	:	HRESULT;	(* HRESULT indicating the result of previous operations (If SUCCEEDED(hrPrev) equals false, no operation is executed.) *)
	END_VAR

END_FUNCTION

// Functions/Drawing/F_VN_DrawCircularArc

	{attribute 'TcIecLibraryType'}
	{attribute 'external_name' := 'F_VN_DrawCircularArc_GUID_E6366096_FAF4_BD73_7D36_427D6B32A0F8'}
	(* Draws a circular arc. *)
	FUNCTION F_VN_DrawCircularArc : HRESULT
	VAR_IN_OUT
		stCircularArc	:	TcVnCircularArc;	(* Circular arc definition *)
	END_VAR
	VAR_INPUT
		ipDestImage	:	ITcVnImage;	(* Destination image *)
	END_VAR
	VAR_IN_OUT
		aColor	:	TcVnVector4_LREAL;	(* Color *)
	END_VAR
	VAR_INPUT
		nThickness	:	DINT;	(* Line thickness (if negative, the arc is filled) *)
		hrPrev	:	HRESULT;	(* HRESULT indicating the result of previous operations (If SUCCEEDED(hrPrev) equals false, no operation is executed.) *)
	END_VAR

END_FUNCTION

// Functions/Drawing/F_VN_DrawCircularArcExp

	{attribute 'TcIecLibraryType'}
	{attribute 'external_name' := 'F_VN_DrawCircularArcExp_GUID_DDDF2BC5_D3BB_B039_6184_0EA1506CA436'}
	(* Draws a circular arc. (expert function) *)
	FUNCTION F_VN_DrawCircularArcExp : HRESULT
	VAR_IN_OUT
		stCircularArc	:	TcVnCircularArc;	(* Circular arc definition *)
	END_VAR
	VAR_INPUT
		ipDestImage	:	ITcVnImage;	(* Destination image *)
	END_VAR
	VAR_IN_OUT
		aColor	:	TcVnVector4_LREAL;	(* Color *)
	END_VAR
	VAR_INPUT
		nThickness	:	DINT;	(* Line thickness (if negative, the arc is filled) *)
		eLineType	:	ETcVnLineType;	(* Line type *)
		hrPrev	:	HRESULT;	(* HRESULT indicating the result of previous operations (If SUCCEEDED(hrPrev) equals false, no operation is executed.) *)
	END_VAR

END_FUNCTION

// Functions/Drawing/F_VN_DrawComponents

	{attribute 'TcIecLibraryType'}
	{attribute 'external_name' := 'F_VN_DrawComponents_GUID_EDFE73EE_D642_B199_78DB_F30E2E307097'}
	(* Draw the results of connected component function. *)
	FUNCTION F_VN_DrawComponents : HRESULT
	VAR_INPUT
		ipLabelImage	:	ITcVnImage;	(* Image contains labels for each pixel (1 channel DINT or UINT). *)
		nLabelID	:	DINT;	(* Value of a specific label to be drawn (if negative, all components within the image are drawn) *)
		ipDestImage	:	REFERENCE TO ITcVnImage;	(* Destination image (An appropriate image will be created if required. The output image is 1 or 3 channels USINT). *)
		bShowLabelID	:	BOOL;	(* Show label ID in the center of the component on the destination image *)
		hrPrev	:	HRESULT;	(* HRESULT indicating the result of previous operations (If SUCCEEDED(hrPrev) equals false, no operation is executed.) *)
	END_VAR

END_FUNCTION

// Functions/Drawing/F_VN_DrawComponentsExp

	{attribute 'TcIecLibraryType'}
	{attribute 'external_name' := 'F_VN_DrawComponentsExp_GUID_639BF640_053E_B917_7759_FC67F1AF1EE2'}
	(* Draw the results of connected component function. (expert function) *)
	FUNCTION F_VN_DrawComponentsExp : HRESULT
	VAR_INPUT
		ipLabelImage	:	ITcVnImage;	(* Image contains labels for each pixel (1 channel DINT or UINT). *)
		nLabelID	:	DINT;	(* Value of a specific label to be drawn (if negative, all components within the image are drawn) *)
		ipDestImage	:	REFERENCE TO ITcVnImage;	(* Destination image (An appropriate image will be created if required. The output image is 1 or 3 channels USINT). *)
		bShowLabelID	:	BOOL;	(* Show lable ID in the center of the component on the destination image *)
	END_VAR
	VAR_IN_OUT
		aColor	:	TcVnVector4_LREAL;	(* Color to draw the components (for {-1, -1, -1, -1}, a random color is chosen for each component) *)
	END_VAR
	VAR_INPUT
		nThickness	:	DINT;	(* Text line thickness *)
		fFontScale	:	LREAL;	(* Scaling factor for the text *)
		hrPrev	:	HRESULT;	(* HRESULT indicating the result of previous operations (If SUCCEEDED(hrPrev) equals false, no operation is executed.) *)
	END_VAR

END_FUNCTION

// Functions/Drawing/F_VN_DrawContours

	{attribute 'TcIecLibraryType'}
	{attribute 'external_name' := 'F_VN_DrawContours_GUID_B9FAF796_61D2_BD69_7C5E_922E4EE577E0'}
	(* Draws a single point set or multiple point sets that are interpreted as contours. *)
	FUNCTION F_VN_DrawContours : HRESULT
	VAR_INPUT
		ipContours	:	ITcVnContainer;	(* Single contour (ContainerType_Vector_TcVnPoint2_DINT) or multiple contours (ContainerType_Vector_Vector_TcVnPoint2_DINT) *)
		nContourIndex	:	DINT;	(* Index of a specific contour to be drawn (if negative, all contours within the container are drawn) *)
		ipDestImage	:	ITcVnImage;	(* Destination image *)
	END_VAR
	VAR_IN_OUT
		aColor	:	TcVnVector4_LREAL;	(* Color *)
	END_VAR
	VAR_INPUT
		nThickness	:	DINT;	(* Line thickness (if negative, the contours are filled) *)
		hrPrev	:	HRESULT;	(* HRESULT indicating the result of previous operations (If SUCCEEDED(hrPrev) equals false, no operation is executed.) *)
	END_VAR

END_FUNCTION

// Functions/Drawing/F_VN_DrawContoursExp

	{attribute 'TcIecLibraryType'}
	{attribute 'external_name' := 'F_VN_DrawContoursExp_GUID_CA97A753_D293_B98B_60CB_153376CD5B38'}
	(* Draws a single point set or multiple point sets that are interpreted as contours. (expert function) *)
	FUNCTION F_VN_DrawContoursExp : HRESULT
	VAR_INPUT
		ipContours	:	ITcVnContainer;	(* Single contour (ContainerType_Vector_TcVnPoint2_DINT) or multiple contours (ContainerType_Vector_Vector_TcVnPoint2_DINT) *)
		nContourIndex	:	DINT;	(* Index of a specific contour to be drawn (if negative, all contours within the container are drawn) *)
		ipDestImage	:	ITcVnImage;	(* Destination image *)
	END_VAR
	VAR_IN_OUT
		aColor	:	TcVnVector4_LREAL;	(* Color *)
	END_VAR
	VAR_INPUT
		nThickness	:	DINT;	(* Line thickness (if negative, the contours are filled) *)
		eLineType	:	ETcVnLineType;	(* Line type *)
		ipHierarchy	:	ITcVnContainer;	(* Contour hierarchy (ContainerType_Vector_TcVnVector4_DINT) *)
		nMaxLevel	:	DINT;	(* Maximum level of contours to be drawn *)
	END_VAR
	VAR_IN_OUT
		aOffset	:	TcVnPoint;	(* Offset by which every contour point is shifted *)
	END_VAR
	VAR_INPUT
		hrPrev	:	HRESULT;	(* HRESULT indicating the result of previous operations (If SUCCEEDED(hrPrev) equals false, no operation is executed.) *)
	END_VAR

END_FUNCTION

// Functions/Drawing/F_VN_DrawEllipse

	{attribute 'TcIecLibraryType'}
	{attribute 'external_name' := 'F_VN_DrawEllipse_GUID_30E759D1_E43E_B2AC_6B7A_71AC013327B2'}
	(* Draws an ellipse. *)
	FUNCTION F_VN_DrawEllipse : HRESULT
	VAR_IN_OUT
		stEllipse	:	TcVnRotatedRectangle;	(* Ellipse to be drawn (rotation angle in degrees) *)
	END_VAR
	VAR_INPUT
		ipDestImage	:	ITcVnImage;	(* Destination image *)
	END_VAR
	VAR_IN_OUT
		aColor	:	TcVnVector4_LREAL;	(* Color *)
	END_VAR
	VAR_INPUT
		nThickness	:	DINT;	(* Line thickness (if negative, the ellipse is filled) *)
		hrPrev	:	HRESULT;	(* HRESULT indicating the result of previous operations (If SUCCEEDED(hrPrev) equals false, no operation is executed.) *)
	END_VAR

END_FUNCTION

// Functions/Drawing/F_VN_DrawEllipseExp

	{attribute 'TcIecLibraryType'}
	{attribute 'external_name' := 'F_VN_DrawEllipseExp_GUID_C1EBC99D_2608_B4C4_4D4D_2FE058324C62'}
	(* Draws an ellipse. (expert function) *)
	FUNCTION F_VN_DrawEllipseExp : HRESULT
	VAR_IN_OUT
		stEllipse	:	TcVnRotatedRectangle;	(* Ellipse to be drawn (rotation angle in degrees) *)
	END_VAR
	VAR_INPUT
		ipDestImage	:	ITcVnImage;	(* Destination image *)
	END_VAR
	VAR_IN_OUT
		aColor	:	TcVnVector4_LREAL;	(* Color *)
	END_VAR
	VAR_INPUT
		nThickness	:	DINT;	(* Line thickness (if negative, the ellipse is filled) *)
		eLineType	:	ETcVnLineType;	(* Line type *)
		hrPrev	:	HRESULT;	(* HRESULT indicating the result of previous operations (If SUCCEEDED(hrPrev) equals false, no operation is executed.) *)
	END_VAR

END_FUNCTION

// Functions/Drawing/F_VN_DrawKeypoints

	{attribute 'TcIecLibraryType'}
	{attribute 'external_name' := 'F_VN_DrawKeypoints_GUID_78B414A4_281B_B6B1_63C8_D29C0654874C'}
	(* Draws the keypoints for visualization purpose. *)
	FUNCTION F_VN_DrawKeypoints : HRESULT
	VAR_INPUT
		ipSrcImage	:	ITcVnImage;	(* Source image (elements of type USINT) *)
		ipKeyPoints	:	ITcVnContainer;	(* Container with the keypoints (ContainerType_Vector_TcVnKeyPoint) *)
		ipDestImage	:	REFERENCE TO ITcVnImage;	(* Destination image (An appropriate color image will be created if required.) *)
		hrPrev	:	HRESULT;	(* HRESULT indicating the result of previous operations (If SUCCEEDED(hrPrev) equals false, no operation is executed.) *)
	END_VAR

END_FUNCTION

// Functions/Drawing/F_VN_DrawKeypointsExp

	{attribute 'TcIecLibraryType'}
	{attribute 'external_name' := 'F_VN_DrawKeypointsExp_GUID_D69F99CA_9EB1_B672_5E38_0A24F0F42CDB'}
	(* Draws the keypoints for visualization purpose. (expert function) *)
	FUNCTION F_VN_DrawKeypointsExp : HRESULT
	VAR_INPUT
		ipSrcImage	:	ITcVnImage;	(* Source image (elements of type USINT) *)
		ipKeyPoints	:	ITcVnContainer;	(* Container with the keypoints (ContainerType_Vector_TcVnKeyPoint) *)
		ipDestImage	:	REFERENCE TO ITcVnImage;	(* Destination image (An appropriate color image will be created if required.) *)
	END_VAR
	VAR_IN_OUT
		aColor	:	TcVnVector4_LREAL;	(* Color to draw the keypoints (for {-1, -1, -1, -1}, a random color is chosen for each point) *)
	END_VAR
	VAR_INPUT
		eFlags	:	ETcVnDrawMatchesFlags;	(* A combination of flags to support overdrawing an existing destination image and/or drawing additional (Rich-)Keypoint information (size and orientation) *)
		hrPrev	:	HRESULT;	(* HRESULT indicating the result of previous operations (If SUCCEEDED(hrPrev) equals false, no operation is executed.) *)
	END_VAR

END_FUNCTION

// Functions/Drawing/F_VN_DrawLine

	{attribute 'TcIecLibraryType'}
	{attribute 'external_name' := 'F_VN_DrawLine_GUID_061C717D_E340_BC7B_58AB_4F85FD18DD44'}
	(* Draws a line. *)
	FUNCTION F_VN_DrawLine : HRESULT
	VAR_INPUT
		nX1	:	UDINT;	(* x coordinate of the start point *)
		nY1	:	UDINT;	(* y coordinate of the start point *)
		nX2	:	UDINT;	(* x coordinate of the end point *)
		nY2	:	UDINT;	(* y coordinate of the end point *)
		ipDestImage	:	ITcVnImage;	(* Destination image *)
	END_VAR
	VAR_IN_OUT
		aColor	:	TcVnVector4_LREAL;	(* Color *)
	END_VAR
	VAR_INPUT
		nThickness	:	DINT;	(* Line thickness *)
		hrPrev	:	HRESULT;	(* HRESULT indicating the result of previous operations (If SUCCEEDED(hrPrev) equals false, no operation is executed.) *)
	END_VAR

END_FUNCTION

// Functions/Drawing/F_VN_DrawLineExp

	{attribute 'TcIecLibraryType'}
	{attribute 'external_name' := 'F_VN_DrawLineExp_GUID_5E4C369F_CA29_BF58_7538_5814068457DF'}
	(* Draws a line. (expert function) *)
	FUNCTION F_VN_DrawLineExp : HRESULT
	VAR_INPUT
		nX1	:	UDINT;	(* x coordinate of the start point *)
		nY1	:	UDINT;	(* y coordinate of the start point *)
		nX2	:	UDINT;	(* x coordinate of the end point *)
		nY2	:	UDINT;	(* y coordinate of the end point *)
		ipDestImage	:	ITcVnImage;	(* Destination image *)
	END_VAR
	VAR_IN_OUT
		aColor	:	TcVnVector4_LREAL;	(* Color *)
	END_VAR
	VAR_INPUT
		nThickness	:	DINT;	(* Line thickness *)
		eLineType	:	ETcVnLineType;	(* Line type *)
		nShift	:	UDINT;	(* Fractional bits of the coordinates (bit shift) *)
		hrPrev	:	HRESULT;	(* HRESULT indicating the result of previous operations (If SUCCEEDED(hrPrev) equals false, no operation is executed.) *)
	END_VAR

END_FUNCTION

// Functions/Drawing/F_VN_DrawLine_TcVnVector4_DINT

	{attribute 'TcIecLibraryType'}
	{attribute 'external_name' := 'F_VN_DrawLine_TcVnVector4_DINT_GUID_88468CA6_43F3_BF6F_598F_301DFE063F24'}
	(* Draws a line. *)
	FUNCTION F_VN_DrawLine_TcVnVector4_DINT : HRESULT
	VAR_IN_OUT
		aLine	:	TcVnVector4_DINT;	(* The start and end point of a line segment [x1, y1, x2, y2] *)
	END_VAR
	VAR_INPUT
		ipDestImage	:	ITcVnImage;	(* Destination image *)
	END_VAR
	VAR_IN_OUT
		aColor	:	TcVnVector4_LREAL;	(* Color *)
	END_VAR
	VAR_INPUT
		nThickness	:	DINT;	(* Line thickness *)
		hrPrev	:	HRESULT;	(* HRESULT indicating the result of previous operations (If SUCCEEDED(hrPrev) equals false, no operation is executed.) *)
	END_VAR

END_FUNCTION

// Functions/Drawing/F_VN_DrawLineExp_TcVnVector4_DINT

	{attribute 'TcIecLibraryType'}
	{attribute 'external_name' := 'F_VN_DrawLineExp_TcVnVector4_DINT_GUID_E828D18A_A6A9_B723_55B6_3C3722406822'}
	(* Draws a line. (expert function) *)
	FUNCTION F_VN_DrawLineExp_TcVnVector4_DINT : HRESULT
	VAR_IN_OUT
		aLine	:	TcVnVector4_DINT;	(* The start and end point of a line segment [x1, y1, x2, y2] *)
	END_VAR
	VAR_INPUT
		ipDestImage	:	ITcVnImage;	(* Destination image *)
	END_VAR
	VAR_IN_OUT
		aColor	:	TcVnVector4_LREAL;	(* Color *)
	END_VAR
	VAR_INPUT
		nThickness	:	DINT;	(* Line thickness *)
		eLineType	:	ETcVnLineType;	(* Line type *)
		nShift	:	UDINT;	(* Fractional bits of the coordinates (bit shift) *)
		hrPrev	:	HRESULT;	(* HRESULT indicating the result of previous operations (If SUCCEEDED(hrPrev) equals false, no operation is executed.) *)
	END_VAR

END_FUNCTION

// Functions/Drawing/F_VN_DrawLine_TcVnVector4_LREAL

	{attribute 'TcIecLibraryType'}
	{attribute 'external_name' := 'F_VN_DrawLine_TcVnVector4_LREAL_GUID_7398C45A_C4BB_B6A9_6287_C45118C963C1'}
	(* Draws a line. *)
	FUNCTION F_VN_DrawLine_TcVnVector4_LREAL : HRESULT
	VAR_IN_OUT
		aLine	:	TcVnVector4_LREAL;	(* The first and second element describe the x and y component of the direction vector. The third and fourth element describe the x and y component of the position vector. *)
	END_VAR
	VAR_INPUT
		ipDestImage	:	ITcVnImage;	(* Destination image *)
	END_VAR
	VAR_IN_OUT
		aColor	:	TcVnVector4_LREAL;	(* Color *)
	END_VAR
	VAR_INPUT
		nThickness	:	DINT;	(* Line thickness *)
		hrPrev	:	HRESULT;	(* HRESULT indicating the result of previous operations (If SUCCEEDED(hrPrev) equals false, no operation is executed.) *)
	END_VAR

END_FUNCTION

// Functions/Drawing/F_VN_DrawLineExp_TcVnVector4_LREAL

	{attribute 'TcIecLibraryType'}
	{attribute 'external_name' := 'F_VN_DrawLineExp_TcVnVector4_LREAL_GUID_CAF1D39B_3754_B79F_61CE_00B3D0FD38CC'}
	(* Draws a line. (expert function) *)
	FUNCTION F_VN_DrawLineExp_TcVnVector4_LREAL : HRESULT
	VAR_IN_OUT
		aLine	:	TcVnVector4_LREAL;	(* The first and second element describe the x and y component of the direction vector. The third and fourth element describe the x and y component of the position vector. *)
	END_VAR
	VAR_INPUT
		ipDestImage	:	ITcVnImage;	(* Destination image *)
	END_VAR
	VAR_IN_OUT
		aColor	:	TcVnVector4_LREAL;	(* Color *)
	END_VAR
	VAR_INPUT
		nThickness	:	DINT;	(* Line thickness *)
		eLineType	:	ETcVnLineType;	(* Line type *)
		nShift	:	UDINT;	(* Fractional bits of the coordinates (bit shift) *)
		hrPrev	:	HRESULT;	(* HRESULT indicating the result of previous operations (If SUCCEEDED(hrPrev) equals false, no operation is executed.) *)
	END_VAR

END_FUNCTION

// Functions/Drawing/F_VN_DrawLines

	{attribute 'TcIecLibraryType'}
	{attribute 'external_name' := 'F_VN_DrawLines_GUID_FC7B078E_1AA4_B750_67FE_2BC7F3E95BE9'}
	(* Draws lines. *)
	FUNCTION F_VN_DrawLines : HRESULT
	VAR_INPUT
		ipLines	:	ITcVnContainer;	(* Container with line descriptions (ContainerType_Vector_TcVnVector2_REAL: the distance from the origin [0] in pixels and the rotation angle [1] in radians. ContainerType_Vector_TcVnVector4_LREAL: the first and second element describe the x and y component of a vector collinear to the line. The third and fourth element describe the x and y component of a point on the line. ContainerType_Vector_TcVnVector4_DINT: start and end point [x1, y1, x2, y2]) *)
		nLineIndex	:	DINT;	(* Index of a specific line to be drawn (if negative, all lines within the container are drawn) *)
		ipDestImage	:	ITcVnImage;	(* Destination image *)
	END_VAR
	VAR_IN_OUT
		aColor	:	TcVnVector4_LREAL;	(* Color *)
	END_VAR
	VAR_INPUT
		nThickness	:	DINT;	(* Line thickness *)
		hrPrev	:	HRESULT;	(* HRESULT indicating the result of previous operations (If SUCCEEDED(hrPrev) equals false, no operation is executed.) *)
	END_VAR

END_FUNCTION

// Functions/Drawing/F_VN_DrawLinesExp

	{attribute 'TcIecLibraryType'}
	{attribute 'external_name' := 'F_VN_DrawLinesExp_GUID_C768A755_451A_B607_778F_A41EBA00D0DB'}
	(* Draws lines. (expert function) *)
	FUNCTION F_VN_DrawLinesExp : HRESULT
	VAR_INPUT
		ipLines	:	ITcVnContainer;	(* Container with line descriptions (ContainerType_Vector_TcVnVector2_REAL: the distance from the origin [0] in pixels and the rotation angle [1] in radians. ContainerType_Vector_TcVnVector4_LREAL: the first and second element describe the x and y component of a vector collinear to the line. The third and fourth element describe the x and y component of a point on the line. ContainerType_Vector_TcVnVector4_DINT: start and end point [x1, y1, x2, y2]) *)
		nLineIndex	:	DINT;	(* Index of a specific line to be drawn (if negative, all lines within the container are drawn) *)
		ipDestImage	:	ITcVnImage;	(* Destination image *)
	END_VAR
	VAR_IN_OUT
		aColor	:	TcVnVector4_LREAL;	(* Color *)
	END_VAR
	VAR_INPUT
		nThickness	:	DINT;	(* Line thickness *)
		eLineType	:	ETcVnLineType;	(* Line type *)
		nShift	:	UDINT;	(* Fractional bits of the coordinates (bit shift) *)
		hrPrev	:	HRESULT;	(* HRESULT indicating the result of previous operations (If SUCCEEDED(hrPrev) equals false, no operation is executed.) *)
	END_VAR

END_FUNCTION

// Functions/Drawing/F_VN_DrawMatches

	{attribute 'TcIecLibraryType'}
	{attribute 'external_name' := 'F_VN_DrawMatches_GUID_17A62AC9_A440_B6CD_4D1A_1995A61BFE13'}
	(* Draws the keypoints and matches for visualization purpose. *)
	FUNCTION F_VN_DrawMatches : HRESULT
	VAR_INPUT
		ipSrcImage1	:	ITcVnImage;	(* Source image 1 (elements of type USINT) *)
		ipKeyPoints1	:	ITcVnContainer;	(* Container with the keypoints 1 (ContainerType_Vector_TcVnKeyPoint) *)
		ipSrcImage2	:	ITcVnImage;	(* Source image 2 (elements of type USINT, must have the same number of channels as ipSrcImage1) *)
		ipKeyPoints2	:	ITcVnContainer;	(* Container with the keypoints 2 (ContainerType_Vector_TcVnKeyPoint) *)
		ipMatches1To2	:	ITcVnContainer;	(* Container with the descriptor matches (ContainerType_Vector_TcVnDMatch) *)
		ipDestImage	:	REFERENCE TO ITcVnImage;	(* Destination image (An appropriate color image will be created if required.) *)
		hrPrev	:	HRESULT;	(* HRESULT indicating the result of previous operations (If SUCCEEDED(hrPrev) equals false, no operation is executed.) *)
	END_VAR

END_FUNCTION

// Functions/Drawing/F_VN_DrawMatchesExp

	{attribute 'TcIecLibraryType'}
	{attribute 'external_name' := 'F_VN_DrawMatchesExp_GUID_5D1F4BA1_221B_B61D_55F1_4C5A260C7288'}
	(* Draws the keypoints and matches for visualization purpose. (expert function) *)
	FUNCTION F_VN_DrawMatchesExp : HRESULT
	VAR_INPUT
		ipSrcImage1	:	ITcVnImage;	(* Source image 1 (elements of type USINT) *)
		ipKeyPoints1	:	ITcVnContainer;	(* Container with the keypoints 1 (ContainerType_Vector_TcVnKeyPoint) *)
		ipSrcImage2	:	ITcVnImage;	(* Source image 2 (elements of type USINT, must have the same number of channels as ipSrcImage1) *)
		ipKeyPoints2	:	ITcVnContainer;	(* Container with the keypoints 2 (ContainerType_Vector_TcVnKeyPoint) *)
		ipMatches1To2	:	ITcVnContainer;	(* Container with the descriptor matches (ContainerType_Vector_TcVnDMatch) *)
		ipDestImage	:	REFERENCE TO ITcVnImage;	(* Destination image (An appropriate color image will be created if required.) *)
	END_VAR
	VAR_IN_OUT
		aMatchColor	:	TcVnVector4_LREAL;	(* Color to draw the matches (for {-1, -1, -1, -1}, a random color is chosen for each point and line) *)
		aSingleColor	:	TcVnVector4_LREAL;	(* Color to draw the single keypoints (for {-1, -1, -1, -1}, a random color is chosen for each point) *)
	END_VAR
	VAR_INPUT
		ipMatchesMask	:	ITcVnContainer;	(* Mask to select the matches to be drawn (ContainerType_Vector_SINT; Set to 0 if all matches should be drawn.) *)
		eFlags	:	ETcVnDrawMatchesFlags;	(* A combination of flags to support overdrawing an existing destination image and/or drawing additional (Rich-)Keypoint information (size and orientation) and/or skipping single keypoints *)
		hrPrev	:	HRESULT;	(* HRESULT indicating the result of previous operations (If SUCCEEDED(hrPrev) equals false, no operation is executed.) *)
	END_VAR

END_FUNCTION

// Functions/Drawing/F_VN_DrawOrientation

	{attribute 'TcIecLibraryType'}
	{attribute 'external_name' := 'F_VN_DrawOrientation_GUID_17DD8F64_54D1_B3E3_563E_1AD0FE64C49E'}
	(* Draw the main axis of a set of points/contour based on a rotated rectangle. *)
	FUNCTION F_VN_DrawOrientation : HRESULT
	VAR_IN_OUT
		stOrientation	:	TcVnRotatedRectangle;	(* Rotated rectangle, containig center of mass, lenghts of axes, and rotation angle in clockwise direction *)
	END_VAR
	VAR_INPUT
		ipDestImage	:	ITcVnImage;	(* Destination image *)
	END_VAR
	VAR_IN_OUT
		aColorMainAxis	:	TcVnVector4_LREAL;	(* Color of the major axis *)
	END_VAR
	VAR_INPUT
		nThickness	:	DINT;	(* Line thickness *)
		hrPrev	:	HRESULT;	(* HRESULT indicating the result of previous operations (If SUCCEEDED(hrPrev) equals false, no operation is executed.) *)
	END_VAR

END_FUNCTION

// Functions/Drawing/F_VN_DrawOrientationExp

	{attribute 'TcIecLibraryType'}
	{attribute 'external_name' := 'F_VN_DrawOrientationExp_GUID_F2EDF790_56AD_B90C_6233_F5B6879E7E70'}
	(* Draw the main axis, the horizontal axis and the angle of a set of points/contour based on a rotated rectangle. (expert function) *)
	FUNCTION F_VN_DrawOrientationExp : HRESULT
	VAR_IN_OUT
		stOrientation	:	TcVnRotatedRectangle;	(* Rotated rectangle, containig center of mass, lenghts of axes, and rotation angle in clockwise direction *)
	END_VAR
	VAR_INPUT
		ipDestImage	:	ITcVnImage;	(* Destination image *)
	END_VAR
	VAR_IN_OUT
		aColorMainAxis	:	TcVnVector4_LREAL;	(* Color of the major axis *)
	END_VAR
	VAR_INPUT
		nThickness	:	DINT;	(* Line thickness *)
	END_VAR
	VAR_IN_OUT
		aColorHorizontalAxis	:	TcVnVector4_LREAL;	(* Color of the horizontal axis *)
	END_VAR
	VAR_INPUT
		fFontScale	:	LREAL;	(* Scaling factor for the text *)
		hrPrev	:	HRESULT;	(* HRESULT indicating the result of previous operations (If SUCCEEDED(hrPrev) equals false, no operation is executed.) *)
	END_VAR

END_FUNCTION

// Functions/Drawing/F_VN_DrawPoint

	{attribute 'TcIecLibraryType'}
	{attribute 'external_name' := 'F_VN_DrawPoint_GUID_70983A07_D591_B08E_77CE_2E6B33EB9ED0'}
	(* Draws a point. *)
	FUNCTION F_VN_DrawPoint : HRESULT
	VAR_INPUT
		nX	:	UDINT;	(* x coordinate of the point *)
		nY	:	UDINT;	(* y coordinate of the point *)
		ipDestImage	:	ITcVnImage;	(* Destination image *)
		eShape	:	ETcVnDrawShape;	(* Point shape *)
	END_VAR
	VAR_IN_OUT
		aColor	:	TcVnVector4_LREAL;	(* Color (for {-1, -1, -1, -1}, a random color is chosen) *)
	END_VAR
	VAR_INPUT
		hrPrev	:	HRESULT;	(* HRESULT indicating the result of previous operations (If SUCCEEDED(hrPrev) equals false, no operation is executed.) *)
	END_VAR

END_FUNCTION

// Functions/Drawing/F_VN_DrawPointExp

	{attribute 'TcIecLibraryType'}
	{attribute 'external_name' := 'F_VN_DrawPointExp_GUID_9730AE5B_BB78_B934_48D1_166F693E5363'}
	(* Draw a point. (expert function) *)
	FUNCTION F_VN_DrawPointExp : HRESULT
	VAR_INPUT
		nX	:	UDINT;	(* x coordinate of the point *)
		nY	:	UDINT;	(* y coordinate of the point *)
		ipDestImage	:	ITcVnImage;	(* Destination image *)
		eShape	:	ETcVnDrawShape;	(* Point shape *)
	END_VAR
	VAR_IN_OUT
		aColor	:	TcVnVector4_LREAL;	(* Color (for {-1, -1, -1, -1}, a random color is chosen) *)
	END_VAR
	VAR_INPUT
		nSize	:	UDINT;	(* Size of the shape (half width) *)
		nThickness	:	DINT;	(* Line thickness (if negative, the shape is filled if it is closed) *)
		eLineType	:	ETcVnLineType;	(* Line type *)
		hrPrev	:	HRESULT;	(* HRESULT indicating the result of previous operations (If SUCCEEDED(hrPrev) equals false, no operation is executed.) *)
	END_VAR

END_FUNCTION

// Functions/Drawing/F_VN_DrawPoints

	{attribute 'TcIecLibraryType'}
	{attribute 'external_name' := 'F_VN_DrawPoints_GUID_7D497842_B7A7_B9D6_5E7B_C0C8A2D39FD1'}
	(* Draw a collection of points. *)
	FUNCTION F_VN_DrawPoints : HRESULT
	VAR_INPUT
		ipPoints	:	ITcVnContainer;	(* Container with TcVnPoint2_DINT or TcVnPoint2_REAL elements *)
		ipDestImage	:	ITcVnImage;	(* Destination image *)
		eShape	:	ETcVnDrawShape;	(* Point shape *)
	END_VAR
	VAR_IN_OUT
		aColor	:	TcVnVector4_LREAL;	(* Color (for {-1, -1, -1, -1}, a random color is chosen for each point) *)
	END_VAR
	VAR_INPUT
		hrPrev	:	HRESULT;	(* HRESULT indicating the result of previous operations (If SUCCEEDED(hrPrev) equals false, no operation is executed.) *)
	END_VAR

END_FUNCTION

// Functions/Drawing/F_VN_DrawPointsExp

	{attribute 'TcIecLibraryType'}
	{attribute 'external_name' := 'F_VN_DrawPointsExp_GUID_AF33D796_B82C_BBA8_4E89_212462C9C118'}
	(* Draw a collection of points. (expert function) *)
	FUNCTION F_VN_DrawPointsExp : HRESULT
	VAR_INPUT
		ipPoints	:	ITcVnContainer;	(* Container with TcVnPoint2_DINT or TcVnPoint2_REAL elements *)
		ipDestImage	:	ITcVnImage;	(* Destination image *)
		eShape	:	ETcVnDrawShape;	(* Point shape *)
	END_VAR
	VAR_IN_OUT
		aColor	:	TcVnVector4_LREAL;	(* Color (for {-1, -1, -1, -1}, a random color is chosen for each point) *)
	END_VAR
	VAR_INPUT
		nSize	:	UDINT;	(* Size of the shape (half width) *)
		nThickness	:	DINT;	(* Line thickness (if negative, the shape is filled if it is closed) *)
		eLineType	:	ETcVnLineType;	(* Line type *)
		hrPrev	:	HRESULT;	(* HRESULT indicating the result of previous operations (If SUCCEEDED(hrPrev) equals false, no operation is executed.) *)
	END_VAR

END_FUNCTION

// Functions/Drawing/F_VN_DrawPolygon

	{attribute 'TcIecLibraryType'}
	{attribute 'external_name' := 'F_VN_DrawPolygon_GUID_B142979D_B57D_BA51_4B71_F7C0BC457F76'}
	(* Draw a pologon using collection of points. *)
	FUNCTION F_VN_DrawPolygon : HRESULT
	VAR_INPUT
		ipPoints	:	ITcVnContainer;	(* Container with TcVnPoint2_DINT, TcVnPoint2_REAL, or TcVnPoint2_LREAL elements *)
		ipDestImage	:	ITcVnImage;	(* Destination image *)
	END_VAR
	VAR_IN_OUT
		aColor	:	TcVnVector4_LREAL;	(* Color *)
	END_VAR
	VAR_INPUT
		nThickness	:	DINT;	(* Line thickness (if negative, the polygon is filled) *)
		hrPrev	:	HRESULT;	(* HRESULT indicating the result of previous operations (If SUCCEEDED(hrPrev) equals false, no operation is executed.) *)
	END_VAR

END_FUNCTION

// Functions/Drawing/F_VN_DrawPolygonExp

	{attribute 'TcIecLibraryType'}
	{attribute 'external_name' := 'F_VN_DrawPolygonExp_GUID_4C1BD5AA_37C5_B658_4481_B4084BE37003'}
	(* Draw a pologon using collection of points. (expert function) *)
	FUNCTION F_VN_DrawPolygonExp : HRESULT
	VAR_INPUT
		ipPoints	:	ITcVnContainer;	(* Container with TcVnPoint2_DINT, TcVnPoint2_REAL, or TcVnPoint2_LREAL elements *)
		ipDestImage	:	ITcVnImage;	(* Destination image *)
	END_VAR
	VAR_IN_OUT
		aColor	:	TcVnVector4_LREAL;	(* Color *)
	END_VAR
	VAR_INPUT
		nThickness	:	DINT;	(* Line thickness (if negative, the shape is filled) *)
		bIsClosed	:	BOOL;	(* If it is true, the function draws a line from the last point to the first point to close the polygon. *)
		eLineType	:	ETcVnLineType;	(* Line type *)
		nShift	:	UDINT;	(* Fractional bits of the coordinates (bit shift) *)
		hrPrev	:	HRESULT;	(* HRESULT indicating the result of previous operations (If SUCCEEDED(hrPrev) equals false, no operation is executed.) *)
	END_VAR

END_FUNCTION

// Functions/Drawing/F_VN_DrawRectangle

	{attribute 'TcIecLibraryType'}
	{attribute 'external_name' := 'F_VN_DrawRectangle_GUID_51F76060_FBA1_B9D3_520C_4A0D0DD2C8C7'}
	(* Draw a rectangle. *)
	FUNCTION F_VN_DrawRectangle : HRESULT
	VAR_INPUT
		nTopLeftX	:	UDINT;	(* x coordinate of the top left corner *)
		nTopLeftY	:	UDINT;	(* y coordinate of the top left corner *)
		nBottomRightX	:	UDINT;	(* x coordinate of the bottom right corner *)
		nBottomRightY	:	UDINT;	(* y coordinate of the bottom right corner *)
		ipDestImage	:	ITcVnImage;	(* Destination image *)
	END_VAR
	VAR_IN_OUT
		aColor	:	TcVnVector4_LREAL;	(* Color *)
	END_VAR
	VAR_INPUT
		nThickness	:	DINT;	(* Line thickness (if negative, the rectangle is filled) *)
		hrPrev	:	HRESULT;	(* HRESULT indicating the result of previous operations (If SUCCEEDED(hrPrev) equals false, no operation is executed.) *)
	END_VAR

END_FUNCTION

// Functions/Drawing/F_VN_DrawRectangle_TcVnRectangle_DINT

	{attribute 'TcIecLibraryType'}
	{attribute 'external_name' := 'F_VN_DrawRectangle_TcVnRectangle_DINT_GUID_AE1440AA_13A8_B9C1_68EA_4B834777CC1E'}
	(* Draw a rectangle. *)
	FUNCTION F_VN_DrawRectangle_TcVnRectangle_DINT : HRESULT
	VAR_IN_OUT
		stRectangle	:	TcVnRectangle_DINT;	(* Rectangle to be drawn *)
	END_VAR
	VAR_INPUT
		ipDestImage	:	ITcVnImage;	(* Destination image *)
	END_VAR
	VAR_IN_OUT
		aColor	:	TcVnVector4_LREAL;	(* Color *)
	END_VAR
	VAR_INPUT
		nThickness	:	DINT;	(* Line thickness (if negative, the rectangle is filled) *)
		hrPrev	:	HRESULT;	(* HRESULT indicating the result of previous operations (If SUCCEEDED(hrPrev) equals false, no operation is executed.) *)
	END_VAR

END_FUNCTION

// Functions/Drawing/F_VN_DrawRectangle_TcVnRectangle_UDINT

	{attribute 'TcIecLibraryType'}
	{attribute 'external_name' := 'F_VN_DrawRectangle_TcVnRectangle_UDINT_GUID_D0F34555_8FD1_BB61_6CC3_A041EA946DEB'}
	(* Draw a rectangle. *)
	FUNCTION F_VN_DrawRectangle_TcVnRectangle_UDINT : HRESULT
	VAR_IN_OUT
		stRectangle	:	TcVnRectangle_UDINT;	(* Rectangle to be drawn *)
	END_VAR
	VAR_INPUT
		ipDestImage	:	ITcVnImage;	(* Destination image *)
	END_VAR
	VAR_IN_OUT
		aColor	:	TcVnVector4_LREAL;	(* Color *)
	END_VAR
	VAR_INPUT
		nThickness	:	DINT;	(* Line thickness (if negative, the rectangle is filled) *)
		hrPrev	:	HRESULT;	(* HRESULT indicating the result of previous operations (If SUCCEEDED(hrPrev) equals false, no operation is executed.) *)
	END_VAR

END_FUNCTION

// Functions/Drawing/F_VN_DrawRotatedRectangle

	{attribute 'TcIecLibraryType'}
	{attribute 'external_name' := 'F_VN_DrawRotatedRectangle_GUID_729EA757_3EEF_BD77_5C18_C5F8FFCB1F64'}
	(* Draw a rectangle. *)
	FUNCTION F_VN_DrawRotatedRectangle : HRESULT
	VAR_IN_OUT
		stRectangle	:	TcVnRotatedRectangle;	(* Rectangle to be drawn (rotation angle in degrees) *)
	END_VAR
	VAR_INPUT
		ipDestImage	:	ITcVnImage;	(* Destination image *)
	END_VAR
	VAR_IN_OUT
		aColor	:	TcVnVector4_LREAL;	(* Color *)
	END_VAR
	VAR_INPUT
		nThickness	:	DINT;	(* Line thickness (if negative, the rectangle is filled) *)
		hrPrev	:	HRESULT;	(* HRESULT indicating the result of previous operations (If SUCCEEDED(hrPrev) equals false, no operation is executed.) *)
	END_VAR

END_FUNCTION

// Functions/Drawing/F_VN_DrawRotatedRectangleExp

	{attribute 'TcIecLibraryType'}
	{attribute 'external_name' := 'F_VN_DrawRotatedRectangleExp_GUID_65878AD2_C6FE_B08A_57A7_E67187187FB0'}
	(* Draw a rectangle. (expert function) *)
	FUNCTION F_VN_DrawRotatedRectangleExp : HRESULT
	VAR_IN_OUT
		stRectangle	:	TcVnRotatedRectangle;	(* Rectangle to be drawn (rotation angle in degrees) *)
	END_VAR
	VAR_INPUT
		ipDestImage	:	ITcVnImage;	(* Destination image *)
	END_VAR
	VAR_IN_OUT
		aColor	:	TcVnVector4_LREAL;	(* Color *)
	END_VAR
	VAR_INPUT
		nThickness	:	DINT;	(* Line thickness (if negative, the rectangle is filled) *)
		eLineType	:	ETcVnLineType;	(* Line type *)
		hrPrev	:	HRESULT;	(* HRESULT indicating the result of previous operations (If SUCCEEDED(hrPrev) equals false, no operation is executed.) *)
	END_VAR

END_FUNCTION

// Functions/Drawing/F_VN_FillCircle

	{attribute 'TcIecLibraryType'}
	{attribute 'external_name' := 'F_VN_FillCircle_GUID_CC76660C_BBCB_B9E7_6F61_1B8F9764D402'}
	(* Paint a filled circle. *)
	FUNCTION F_VN_FillCircle : HRESULT
	VAR_INPUT
		nCenterX	:	UDINT;	(* x coordinate of the center *)
		nCenterY	:	UDINT;	(* y coordinate of the center *)
		nRadius	:	UDINT;	(* Radius *)
		ipDestImage	:	ITcVnImage;	(* Destination image *)
	END_VAR
	VAR_IN_OUT
		aColor	:	TcVnVector4_LREAL;	(* Color *)
	END_VAR
	VAR_INPUT
		hrPrev	:	HRESULT;	(* HRESULT indicating the result of previous operations (If SUCCEEDED(hrPrev) equals false, no operation is executed.) *)
	END_VAR

END_FUNCTION

// Functions/Drawing/F_VN_FillContours

	{attribute 'TcIecLibraryType'}
	{attribute 'external_name' := 'F_VN_FillContours_GUID_01969524_59A2_B7C2_5DB7_B0C76998DF31'}
	(* Paint a single point set or multiple point sets that are interpreted as contours. *)
	FUNCTION F_VN_FillContours : HRESULT
	VAR_INPUT
		ipContours	:	ITcVnContainer;	(* Single contour (ContainerType_Vector_TcVnPoint2_DINT) or multiple contours (ContainerType_Vector_Vector_TcVnPoint2_DINT) *)
		nContourIndex	:	DINT;	(* Index of a specific contour to be drawn (if negative, all contours within the container are drawn) *)
		ipDestImage	:	ITcVnImage;	(* Destination image *)
	END_VAR
	VAR_IN_OUT
		aColor	:	TcVnVector4_LREAL;	(* Color *)
	END_VAR
	VAR_INPUT
		hrPrev	:	HRESULT;	(* HRESULT indicating the result of previous operations (If SUCCEEDED(hrPrev) equals false, no operation is executed.) *)
	END_VAR

END_FUNCTION

// Functions/Drawing/F_VN_FillEllipse

	{attribute 'TcIecLibraryType'}
	{attribute 'external_name' := 'F_VN_FillEllipse_GUID_C758DDF8_D4B0_BC68_56CE_BB1630168A3B'}
	(* Paint a filled ellipse. *)
	FUNCTION F_VN_FillEllipse : HRESULT
	VAR_IN_OUT
		stEllipse	:	TcVnRotatedRectangle;	(* Ellipse to be painted (rotation angle in degrees) *)
	END_VAR
	VAR_INPUT
		ipDestImage	:	ITcVnImage;	(* Destination image *)
	END_VAR
	VAR_IN_OUT
		aColor	:	TcVnVector4_LREAL;	(* Color *)
	END_VAR
	VAR_INPUT
		hrPrev	:	HRESULT;	(* HRESULT indicating the result of previous operations (If SUCCEEDED(hrPrev) equals false, no operation is executed.) *)
	END_VAR

END_FUNCTION

// Functions/Drawing/F_VN_FillPolygon

	{attribute 'TcIecLibraryType'}
	{attribute 'external_name' := 'F_VN_FillPolygon_GUID_BE4AA06B_560B_BC82_4C3B_26BFD185E222'}
	(* Paint a filled pologon using a set of points. *)
	FUNCTION F_VN_FillPolygon : HRESULT
	VAR_INPUT
		ipPoints	:	ITcVnContainer;	(* Container with TcVnPoint2_DINT, TcVnPoint2_REAL, or TcVnPoint2_LREAL elements *)
		ipDestImage	:	ITcVnImage;	(* Destination image *)
	END_VAR
	VAR_IN_OUT
		aColor	:	TcVnVector4_LREAL;	(* Color *)
	END_VAR
	VAR_INPUT
		hrPrev	:	HRESULT;	(* HRESULT indicating the result of previous operations (If SUCCEEDED(hrPrev) equals false, no operation is executed.) *)
	END_VAR

END_FUNCTION

// Functions/Drawing/F_VN_FillRectangle

	{attribute 'TcIecLibraryType'}
	{attribute 'external_name' := 'F_VN_FillRectangle_GUID_2D7701D6_020C_B985_6A7D_A8B426F4B202'}
	(* Paint a filled rectangle. *)
	FUNCTION F_VN_FillRectangle : HRESULT
	VAR_INPUT
		nTopLeftX	:	UDINT;	(* x coordinate of the top left corner *)
		nTopLeftY	:	UDINT;	(* y coordinate of the top left corner *)
		nBottomRightX	:	UDINT;	(* x coordinate of the bottom right corner *)
		nBottomRightY	:	UDINT;	(* y coordinate of the bottom right corner *)
		ipDestImage	:	ITcVnImage;	(* Destination image *)
	END_VAR
	VAR_IN_OUT
		aColor	:	TcVnVector4_LREAL;	(* Color *)
	END_VAR
	VAR_INPUT
		hrPrev	:	HRESULT;	(* HRESULT indicating the result of previous operations (If SUCCEEDED(hrPrev) equals false, no operation is executed.) *)
	END_VAR

END_FUNCTION

// Functions/Drawing/F_VN_FillRotatedRectangle

	{attribute 'TcIecLibraryType'}
	{attribute 'external_name' := 'F_VN_FillRotatedRectangle_GUID_9E9ADE36_0A41_BB66_564E_0FE623952F15'}
	(* Paint a filled rectangle. *)
	FUNCTION F_VN_FillRotatedRectangle : HRESULT
	VAR_IN_OUT
		stRectangle	:	TcVnRotatedRectangle;	(* Rectangle to be painted (rotation angle in degrees) *)
	END_VAR
	VAR_INPUT
		ipDestImage	:	ITcVnImage;	(* Destination image *)
	END_VAR
	VAR_IN_OUT
		aColor	:	TcVnVector4_LREAL;	(* Color *)
	END_VAR
	VAR_INPUT
		hrPrev	:	HRESULT;	(* HRESULT indicating the result of previous operations (If SUCCEEDED(hrPrev) equals false, no operation is executed.) *)
	END_VAR

END_FUNCTION

// Functions/Drawing/F_VN_PlotIntensityProfile

	{attribute 'TcIecLibraryType'}
	{attribute 'external_name' := 'F_VN_PlotIntensityProfile_GUID_2921089B_8CB7_B726_4E3D_EBC3C94893A8'}
	(* Plots the pixel intensity profile along a line segment in an image. *)
	FUNCTION F_VN_PlotIntensityProfile : HRESULT
	VAR_INPUT
		ipSrcImage	:	ITcVnImage;	(* Source image (USINT, 1 channel) *)
		ipDestImage	:	REFERENCE TO ITcVnImage;	(* Destination image (USINT, 1 channel. x: position, y: intensity, origin: bottom left. An appropriate destination image will be created if required.) *)
	END_VAR
	VAR_IN_OUT
		aStartPoint	:	TcVnPoint2_REAL;	(* Start point of the line segment *)
		aEndPoint	:	TcVnPoint2_REAL;	(* End point of the line segment *)
	END_VAR
	VAR_INPUT
		hrPrev	:	HRESULT;	(* HRESULT indicating the result of previous operations (If SUCCEEDED(hrPrev) equals false, no operation is executed.) *)
	END_VAR

END_FUNCTION

// Functions/Drawing/F_VN_PlotIntensityProfileExp

	{attribute 'TcIecLibraryType'}
	{attribute 'external_name' := 'F_VN_PlotIntensityProfileExp_GUID_835D66C2_F439_B08A_5DBF_25451AFA2CBA'}
	(* Plots the pixel intensity profile along a line segment in an image. (expert function) *)
	FUNCTION F_VN_PlotIntensityProfileExp : HRESULT
	VAR_INPUT
		ipSrcImage	:	ITcVnImage;	(* Source image (USINT, 1 channel) *)
		ipDestImage	:	REFERENCE TO ITcVnImage;	(* Destination image (USINT, 1 channel. x: position, y: intensity, origin: bottom left. An appropriate destination image will be created if required.) *)
	END_VAR
	VAR_IN_OUT
		aStartPoint	:	TcVnPoint2_REAL;	(* Start point of the line segment *)
		aEndPoint	:	TcVnPoint2_REAL;	(* End point of the line segment *)
		aBackgroundColor	:	TcVnVector4_LREAL;	(* Background color *)
		aLineColor	:	TcVnVector4_LREAL;	(* Line color *)
		aGridColor	:	TcVnVector4_LREAL;	(* Grid color *)
	END_VAR
	VAR_INPUT
		nScaleX	:	DINT;	(* Scale in x direction (ipDestImage will have a width of nScaleX * (ipSrcImage width - 1) + 1) *)
		nScaleY	:	DINT;	(* Scale in y direction (ipDestImage will have a height of nScaleY * 255 + 1) *)
		nThickness	:	DINT;	(* Line thickness *)
		nDestChannels	:	DINT;	(* ipDestImage channels (1 or 3) *)
		hrPrev	:	HRESULT;	(* HRESULT indicating the result of previous operations (If SUCCEEDED(hrPrev) equals false, no operation is executed.) *)
	END_VAR

END_FUNCTION

// Functions/Drawing/F_VN_PutLabel

	{attribute 'TcIecLibraryType'}
	{attribute 'external_name' := 'F_VN_PutLabel_GUID_37A07087_02CE_B882_533D_C090C07A4E17'}
	(* Write a label (black text on white background) into an image. *)
	FUNCTION F_VN_PutLabel : HRESULT
	VAR_IN_OUT CONSTANT
		sText	:	STRING;	(* Text *)
	END_VAR
	VAR_INPUT
		ipDestImage	:	ITcVnImage;	(* Destination image *)
		nX	:	UDINT;	(* x coordinate (bottom left) *)
		nY	:	UDINT;	(* y coordinate (bottom left) *)
		fFontScale	:	LREAL;	(* Scaling factor *)
		hrPrev	:	HRESULT;	(* HRESULT indicating the result of previous operations (If SUCCEEDED(hrPrev) equals false, no operation is executed.) *)
	END_VAR

END_FUNCTION

// Functions/Drawing/F_VN_PutLabelExp

	{attribute 'TcIecLibraryType'}
	{attribute 'external_name' := 'F_VN_PutLabelExp_GUID_B9541024_C435_B902_75B0_95E7657E4854'}
	(* Write a label (text on unified background) into an image. (expert function) *)
	FUNCTION F_VN_PutLabelExp : HRESULT
	VAR_IN_OUT CONSTANT
		sText	:	STRING;	(* Text *)
	END_VAR
	VAR_INPUT
		ipDestImage	:	ITcVnImage;	(* Destination image *)
		nX	:	UDINT;	(* x coordinate (bottom left) *)
		nY	:	UDINT;	(* y coordinate (bottom left) *)
		fFontScale	:	LREAL;	(* Scaling factor *)
		nThickness	:	UDINT;	(* Line thickness *)
		eFontType	:	ETcVnFontType;	(* Font type *)
	END_VAR
	VAR_IN_OUT
		aFontColor	:	TcVnVector4_LREAL;	(* Font color *)
		aBackgroundColor	:	TcVnVector4_LREAL;	(* Background color *)
	END_VAR
	VAR_INPUT
		eLineType	:	ETcVnLineType;	(* Line type *)
		hrPrev	:	HRESULT;	(* HRESULT indicating the result of previous operations (If SUCCEEDED(hrPrev) equals false, no operation is executed.) *)
	END_VAR

END_FUNCTION

// Functions/Drawing/F_VN_PutText

	{attribute 'TcIecLibraryType'}
	{attribute 'external_name' := 'F_VN_PutText_GUID_11053B6D_CD68_B7DC_52E3_2F55A81D5517'}
	(* Write text into an image. *)
	FUNCTION F_VN_PutText : HRESULT
	VAR_IN_OUT CONSTANT
		sText	:	STRING;	(* Text *)
	END_VAR
	VAR_INPUT
		ipDestImage	:	ITcVnImage;	(* Destination image *)
		nX	:	UDINT;	(* x coordinate (bottom left) *)
		nY	:	UDINT;	(* y coordinate (bottom left) *)
		eFontType	:	ETcVnFontType;	(* Font type *)
		fFontScale	:	LREAL;	(* Scaling factor *)
	END_VAR
	VAR_IN_OUT
		aColor	:	TcVnVector4_LREAL;	(* Text color *)
	END_VAR
	VAR_INPUT
		hrPrev	:	HRESULT;	(* HRESULT indicating the result of previous operations (If SUCCEEDED(hrPrev) equals false, no operation is executed.) *)
	END_VAR

END_FUNCTION

// Functions/Drawing/F_VN_PutTextExp

	{attribute 'TcIecLibraryType'}
	{attribute 'external_name' := 'F_VN_PutTextExp_GUID_430C51EA_AFCA_B90B_6E89_23858F30F33D'}
	(* Write text into an image. (expert function) *)
	FUNCTION F_VN_PutTextExp : HRESULT
	VAR_IN_OUT CONSTANT
		sText	:	STRING;	(* Text *)
	END_VAR
	VAR_INPUT
		ipDestImage	:	ITcVnImage;	(* Destination image *)
		nX	:	UDINT;	(* x coordinate (bottom left) *)
		nY	:	UDINT;	(* y coordinate (bottom left) *)
		eFontType	:	ETcVnFontType;	(* Font type *)
		fFontScale	:	LREAL;	(* Scaling factor *)
	END_VAR
	VAR_IN_OUT
		aColor	:	TcVnVector4_LREAL;	(* Text color *)
	END_VAR
	VAR_INPUT
		nThickness	:	DINT;	(* Line thickness *)
		eLineType	:	ETcVnLineType;	(* Line type *)
		bBottomLeftOrigin	:	BOOL;	(* Sets the image origin to the bottom left corner, if true *)
		hrPrev	:	HRESULT;	(* HRESULT indicating the result of previous operations (If SUCCEEDED(hrPrev) equals false, no operation is executed.) *)
	END_VAR

END_FUNCTION

// Functions/Keypoint Features/F_VN_FilterGoodMatches

	{attribute 'TcIecLibraryType'}
	{attribute 'external_name' := 'F_VN_FilterGoodMatches_GUID_84217484_78D0_BCC4_7DA2_7B60CECB633F'}
	(* Filter the descriptor matches and return only good ones. *)
	FUNCTION F_VN_FilterGoodMatches : HRESULT
	VAR_INPUT
		ipMatches	:	ITcVnContainer;	(* Container with descriptor matches (ContainerType_Vector_TcVnDMatch or ContainerType_Vector_Vector_TcVnDMatch) *)
		ipGoodMatches	:	REFERENCE TO ITcVnContainer;	(* Returns a container with good matches (ContainerType_Vector_TcVnDMatch) *)
		fMaxDist	:	REAL;	(* Maximum allowed descriptor distance (-1 disables this filter criterion) *)
		fMaxKnnRatio	:	REAL;	(* Maximum allowed distance ratio between first and second best match ([0..1], used for knn match results only, -1 disables this filter criterion) *)
		hrPrev	:	HRESULT;	(* HRESULT indicating the result of previous operations (If SUCCEEDED(hrPrev) equals false, no operation is executed.) *)
	END_VAR

END_FUNCTION

// Functions/Keypoint Features/F_VN_FindReferenceKeyPointsInImage

	{attribute 'TcIecLibraryType'}
	{attribute 'external_name' := 'F_VN_FindReferenceKeyPointsInImage_GUID_8578F0CC_537C_BAAB_643C_A9D296438311'}
	(* Searches a reference image, represented by its keypoints and corresponding descriptors, in a given source image. *)
	FUNCTION F_VN_FindReferenceKeyPointsInImage : HRESULT
	VAR_INPUT
		ipSrcKeyPoints	:	ITcVnContainer;	(* KeyPoints of the source image, e.g. (ContainerType_Vector_TcVnKeyPoint) *)
		ipSrcDescriptors	:	ITcVnImage;	(* Descriptors of the source image KeyPoints *)
		ipRefKeyPoints	:	ITcVnContainer;	(* KeyPoints of the reference image, e.g. (ContainerType_Vector_TcVnKeyPoint) *)
		ipRefDescriptors	:	ITcVnImage;	(* Descriptors of the reference image KeyPoints *)
		nRefImageWidth	:	UDINT;	(* Width of the reference image in pixels *)
		nRefImageHeight	:	UDINT;	(* Height of the reference image in pixels *)
		ipEdgePoints	:	REFERENCE TO ITcVnContainer;	(* Returns a container with the 4 edge points of the reference image transformed into the coordinates of the source image (ContainerType_Vector_TcVnPoint2_REAL) *)
		fMaxDist	:	REAL;	(* Maximum allowed descriptor distance (-1 disables this filter criterion) *)
		fMaxKnnRatio	:	REAL;	(* Maximum allowed distance ratio between first and second best match ([0..1], -1 disables this filter criterion) *)
		eNormType	:	ETcVnNormalizationType;	(* Normalization type used for descriptor matching (HAMMING recommended for AKAZE, ORB, and BRISK. HAMMING2 is recommended for ORB if the ORB nBriefPoints parameter is 3 or 4. ) *)
		hrPrev	:	HRESULT;	(* HRESULT indicating the result of previous operations (If SUCCEEDED(hrPrev) equals false, no operation is executed.) *)
	END_VAR
	VAR_OUTPUT
		aPerspectiveTransform	:	TcVnMatrix3x3_LREAL;	(* Returns the perspective transformation matrix, which transforms the reference points to the source points *)
		nNumberOfGoodMatches	:	UDINT;	(* Return the number of good matches *)
		nNumberOfInliers	:	UDINT;	(* Return the number of inlier matches *)
	END_VAR

END_FUNCTION

// Functions/Keypoint Features/F_VN_FindReferenceKeyPointsInImageExp

	{attribute 'TcIecLibraryType'}
	{attribute 'external_name' := 'F_VN_FindReferenceKeyPointsInImageExp_GUID_C11B0F13_7989_BA6F_58A8_E8003D2A5B03'}
	(* Searches a reference image, represented by its keypoints and corresponding descriptors, in a given source image. (expert function) *)
	FUNCTION F_VN_FindReferenceKeyPointsInImageExp : HRESULT
	VAR_INPUT
		ipSrcKeyPoints	:	ITcVnContainer;	(* KeyPoints of the source image, e.g. (ContainerType_Vector_TcVnKeyPoint) *)
		ipSrcDescriptors	:	ITcVnImage;	(* Descriptors of the source image KeyPoints *)
		ipRefKeyPoints	:	ITcVnContainer;	(* KeyPoints of the reference image (ContainerType_Vector_TcVnKeyPoint) *)
		ipRefDescriptors	:	ITcVnImage;	(* Descriptors of the reference image KeyPoints *)
		nRefImageWidth	:	UDINT;	(* Width of the reference image in pixels *)
		nRefImageHeight	:	UDINT;	(* Height of the reference image in pixels *)
		ipEdgePoints	:	REFERENCE TO ITcVnContainer;	(* Returns a container with the 4 edge points of the reference image transformed into the coordinates of the source image (ContainerType_Vector_TcVnPoint2_REAL) *)
		fMaxDist	:	REAL;	(* Maximum allowed descriptor distance (-1 disables this filter criterion) *)
		fMaxKnnRatio	:	REAL;	(* Maximum allowed distance ratio between first and second best match ([0..1], -1 disables this filter criterion) *)
		eNormType	:	ETcVnNormalizationType;	(* Normalization type used for descriptor matching (HAMMING recommended for AKAZE, ORB, and BRISK. HAMMING2 is recommended for ORB if the ORB nBriefPoints parameter is 3 or 4. ) *)
		eAlgorithm	:	ETcVnEstimationAlgorithm;	(* Estimation algorithm used for computing the perspective transformation between the two point sets *)
		fReprojThreshold	:	LREAL;	(* Maximum allowed reprojection error to treat a point pair as an inlier (only used if eAlgorithm is RANSAC, RHO) *)
		nMaxIterations	:	UDINT;	(* Maximum number of RANSAC iterations *)
		fConfidence	:	LREAL;	(* Confidence (0..1) *)
		ipGoodMatches	:	REFERENCE TO ITcVnContainer;	(* Returns a container with good matches (optional, set to 0 if not required; ContainerType_Vector_TcVnDMatch) *)
		ipInlierMask	:	REFERENCE TO ITcVnContainer;	(* Returns a mask marking the inliers (optional, set to 0 if not required; ContainerType_Vector_SINT; only for RANSAC, LMEDS) *)
		hrPrev	:	HRESULT;	(* HRESULT indicating the result of previous operations (If SUCCEEDED(hrPrev) equals false, no operation is executed.) *)
	END_VAR
	VAR_OUTPUT
		aPerspectiveTransform	:	TcVnMatrix3x3_LREAL;	(* Returns the perspective transformation matrix, which transforms the reference points to the source points  *)
		nNumberOfGoodMatches	:	UDINT;	(* Return the number of good matches *)
		nNumberOfInliers	:	UDINT;	(* Return the number of inlier matches *)
	END_VAR

END_FUNCTION

